C03637=1145.324,-115.065,-43.612,178.627,5.983,149.479
C03638=1145.319,-114.815,-43.621,178.630,5.984,149.478
C03639=1145.313,-114.565,-43.629,178.632,5.984,149.478
C03640=1145.308,-114.315,-43.638,178.634,5.984,149.477
C03641=1145.302,-114.066,-43.647,178.636,5.985,149.477
C03642=1145.297,-113.816,-43.655,178.637,5.985,149.476
C03643=1145.292,-113.566,-43.664,178.640,5.986,149.476
C03644=1145.286,-113.316,-43.672,178.641,5.986,149.475
C03645=1145.281,-113.066,-43.681,178.643,5.986,149.475
C03646=1145.276,-112.816,-43.690,178.646,5.987,149.474
C03647=1145.270,-112.567,-43.699,178.648,5.987,149.473
C03648=1145.265,-112.317,-43.708,178.650,5.988,149.473
C03649=1145.259,-112.068,-43.716,178.651,5.987,149.472
C03650=1145.254,-111.818,-43.725,178.654,5.988,149.472
C03651=1145.249,-111.568,-43.734,178.655,5.988,149.471
C03652=1145.244,-111.317,-43.742,178.657,5.989,149.471
C03653=1145.238,-111.068,-43.751,178.660,5.990,149.470
C03654=1145.232,-110.818,-43.760,178.661,5.990,149.470
C03655=1145.227,-110.568,-43.769,178.664,5.990,149.469
C03656=1145.222,-110.318,-43.778,178.665,5.990,149.469
C03657=1145.217,-110.069,-43.787,178.668,5.991,149.468
C03658=1145.211,-109.819,-43.796,178.669,5.991,149.468
C03659=1145.206,-109.570,-43.804,178.671,5.991,149.467
C03660=1145.200,-109.320,-43.813,178.674,5.992,149.467
C03661=1145.195,-109.070,-43.822,178.675,5.992,149.466
C03662=1145.190,-108.820,-43.831,178.678,5.992,149.466
C03663=1145.185,-108.570,-43.840,178.680,5.992,149.465
C03664=1145.179,-108.321,-43.849,178.682,5.993,149.465
C03665=1145.173,-108.071,-43.858,178.683,5.993,149.464
C03666=1145.168,-107.821,-43.867,178.685,5.994,149.464
C03667=1145.163,-107.571,-43.876,178.688,5.995,149.463
C03668=1145.158,-107.321,-43.885,178.689,5.995,149.463
C03669=1145.153,-107.071,-43.894,178.691,5.995,149.462
C03670=1145.147,-106.822,-43.902,178.694,5.995,149.462
C03671=1145.142,-106.572,-43.911,178.696,5.996,149.461
C03672=1145.136,-106.322,-43.921,178.698,5.996,149.461
C03673=1145.131,-106.072,-43.929,178.700,5.996,149.460
C03674=1145.125,-105.823,-43.938,178.702,5.997,149.460
C03675=1145.120,-105.573,-43.947,178.703,5.997,149.459
C03676=1145.115,-105.323,-43.956,178.706,5.998,149.458
C03677=1145.110,-105.073,-43.965,178.708,5.998,149.458
C03678=1145.103,-104.824,-43.974,178.710,5.998,149.457
C03679=1145.098,-104.574,-43.983,178.712,5.999,149.457
C03680=1145.093,-104.324,-43.992,178.714,5.999,149.456
C03681=1145.088,-104.074,-44.001,178.716,6.000,149.456
C03682=1145.083,-103.824,-44.010,178.718,6.000,149.455
C03683=1145.077,-103.575,-44.020,178.720,6.000,149.455
C03684=1145.072,-103.325,-44.029,178.722,6.001,149.454
C03685=1145.066,-103.052,-44.038,178.724,6.002,149.454
C03686=1145.060,-102.781,-44.048,178.727,6.001,149.453
C03687=1145.054,-102.508,-44.058,178.729,6.002,149.453
C03688=1145.049,-102.237,-44.068,178.731,6.003,149.452
C03689=1145.044,-101.987,-44.077,178.733,6.003,149.452
C03690=1145.038,-101.737,-44.086,178.735,6.003,149.451
C03691=1145.033,-101.487,-44.095,178.737,6.004,149.450
C03692=1145.027,-101.237,-44.104,178.739,6.004,149.450
C03693=1145.023,-100.988,-44.114,178.741,6.004,149.449
C03694=1145.017,-100.737,-44.123,178.743,6.005,149.449
C03695=1145.011,-100.488,-44.132,178.745,6.005,149.448
C03696=1145.006,-100.238,-44.141,178.748,6.005,149.448
C03697=1145.001,-99.989,-44.150,178.749,6.005,149.447
C03698=1144.995,-99.738,-44.159,178.751,6.006,149.447
C03699=1144.990,-99.489,-44.169,178.754,6.007,149.446
C03700=1144.985,-99.239,-44.178,178.755,6.007,149.446
C03701=1144.979,-98.989,-44.187,178.758,6.007,149.445
C03702=1144.974,-98.739,-44.196,178.760,6.008,149.445
C03703=1144.969,-98.490,-44.206,178.762,6.008,149.444
C03704=1144.963,-98.240,-44.215,178.764,6.009,149.444
C03705=1144.958,-97.990,-44.224,178.766,6.010,149.443
C03706=1144.952,-97.740,-44.233,178.768,6.010,149.443
C03707=1144.947,-97.491,-44.243,178.770,6.010,149.442
C03708=1144.942,-97.241,-44.252,178.772,6.010,149.441
C03709=1144.936,-96.991,-44.261,178.774,6.011,149.441
C03710=1144.931,-96.741,-44.270,178.776,6.011,149.441
C03711=1144.926,-96.492,-44.280,178.778,6.011,149.440
C03712=1144.921,-96.242,-44.289,178.781,6.012,149.439
C03713=1144.915,-95.992,-44.298,178.783,6.012,149.439
C03714=1144.909,-95.742,-44.307,178.784,6.012,149.438
C03715=1144.905,-95.492,-44.317,178.787,6.013,149.438
C03716=1144.899,-95.242,-44.326,178.789,6.014,149.437
C03717=1144.894,-94.992,-44.335,178.791,6.013,149.437
C03718=1144.888,-94.743,-44.346,178.793,6.014,149.436
C03719=1144.883,-94.493,-44.354,178.795,6.015,149.436
C03720=1144.878,-94.243,-44.363,178.797,6.015,149.435
C03721=1144.872,-93.994,-44.374,178.799,6.016,149.435
C03722=1144.867,-93.744,-44.382,178.801,6.015,149.434
C03723=1144.862,-93.495,-44.392,178.803,6.016,149.434
C03724=1144.856,-93.244,-44.402,178.806,6.017,149.433
C03725=1144.851,-92.995,-44.410,178.807,6.017,149.433
C03726=1144.845,-92.745,-44.421,178.809,6.018,149.432
C03727=1144.840,-92.495,-44.430,178.812,6.018,149.431
C03728=1144.834,-92.245,-44.439,178.814,6.018,149.431
C03729=1144.829,-91.996,-44.449,178.816,6.019,149.430
C03730=1144.824,-91.746,-44.458,178.818,6.019,149.430
C03731=1144.819,-91.496,-44.468,178.820,6.019,149.429
C03732=1144.813,-91.247,-44.477,178.822,6.020,149.429
C03733=1144.808,-90.997,-44.487,178.824,6.021,149.428
C03734=1144.803,-90.747,-44.496,178.826,6.020,149.428
C03735=1144.797,-90.497,-44.505,178.828,6.021,149.427
C03736=1144.792,-90.248,-44.515,178.831,6.022,149.427
C03737=1144.787,-89.997,-44.525,178.832,6.022,149.426
C03738=1144.782,-89.748,-44.534,178.835,6.022,149.426
C03739=1144.776,-89.497,-44.544,178.837,6.023,149.425
C03740=1144.771,-89.248,-44.553,178.839,6.023,149.424
C03741=1144.765,-88.998,-44.563,178.841,6.023,149.424
C03742=1144.760,-88.749,-44.573,178.843,6.024,149.423
C03743=1144.754,-88.499,-44.582,178.846,6.025,149.423
C03744=1144.749,-88.249,-44.592,178.847,6.025,149.422
C03745=1144.744,-87.999,-44.601,178.850,6.025,149.422
C03746=1144.739,-87.750,-44.611,178.852,6.026,149.421
C03747=1144.733,-87.500,-44.620,178.854,6.026,149.421
C03748=1144.729,-87.250,-44.630,178.856,6.027,149.420
C03749=1144.723,-87.000,-44.640,178.858,6.027,149.420
C03750=1144.718,-86.751,-44.649,178.860,6.027,149.419
C03751=1144.712,-86.501,-44.660,178.862,6.028,149.419
C03752=1144.707,-86.251,-44.668,178.864,6.029,149.418
C03753=1144.701,-86.002,-44.679,178.867,6.028,149.417
C03754=1144.696,-85.752,-44.688,178.869,6.029,149.417
C03755=1144.691,-85.502,-44.698,178.871,6.030,149.416
C03756=1144.686,-85.252,-44.707,178.872,6.030,149.416
C03757=1144.680,-85.002,-44.717,178.875,6.030,149.415
C03758=1144.676,-84.753,-44.727,178.877,6.031,149.415
C03759=1144.670,-84.503,-44.736,178.880,6.032,149.414
C03760=1144.664,-84.253,-44.747,178.881,6.032,149.414
C03761=1144.659,-84.003,-44.755,178.884,6.032,149.413
C03762=1144.653,-83.754,-44.766,178.886,6.033,149.413
C03763=1144.649,-83.504,-44.776,178.888,6.033,149.412
C03764=1144.643,-83.254,-44.785,178.890,6.033,149.412
C03765=1144.638,-83.004,-44.795,178.892,6.034,149.411
C03766=1144.633,-82.755,-44.805,178.894,6.034,149.410
C03767=1144.627,-82.505,-44.814,178.896,6.035,149.410
C03768=1144.622,-82.256,-44.824,178.898,6.035,149.409
C03769=1144.617,-82.005,-44.835,178.901,6.036,149.409
C03770=1144.611,-81.755,-44.844,178.903,6.036,149.408
C03771=1144.606,-81.506,-44.854,178.905,6.036,149.408
C03772=1144.601,-81.256,-44.864,178.907,6.037,149.407
C03773=1144.595,-81.006,-44.873,178.909,6.037,149.407
C03774=1144.590,-80.756,-44.883,178.911,6.038,149.406
C03775=1144.585,-80.507,-44.894,178.914,6.038,149.406
C03776=1144.579,-80.257,-44.904,178.916,6.039,149.405
C03777=1144.574,-80.007,-44.913,178.918,6.039,149.404
C03778=1144.568,-79.758,-44.923,178.920,6.039,149.404
C03779=1144.563,-79.508,-44.934,178.922,6.040,149.403
C03780=1144.559,-79.258,-44.943,178.924,6.041,149.403
C03781=1144.553,-79.008,-44.953,178.926,6.041,149.402
C03782=1144.547,-78.759,-44.963,178.929,6.041,149.402
C03783=1144.542,-78.509,-44.972,178.931,6.042,149.401
C03784=1144.537,-78.259,-44.983,178.933,6.042,149.401
C03785=1144.531,-78.009,-44.993,178.935,6.042,149.400
C03786=1144.526,-77.759,-45.003,178.937,6.043,149.400
C03787=1144.521,-77.510,-45.012,178.940,6.044,149.399
C03788=1144.515,-77.261,-45.023,178.942,6.044,149.398
C03789=1144.509,-76.989,-45.034,178.944,6.044,149.398
C03790=1144.504,-76.717,-45.044,178.946,6.045,149.397
C03791=1144.499,-76.446,-45.055,178.949,6.045,149.397
C03792=1144.492,-76.175,-45.066,178.951,6.046,149.396
C03793=1144.487,-75.925,-45.077,178.954,6.047,149.396
C03794=1144.482,-75.675,-45.086,178.955,6.047,149.395
C03795=1144.476,-75.425,-45.096,178.957,6.047,149.395
C03796=1144.471,-75.176,-45.106,178.960,6.048,149.394
C03797=1144.466,-74.926,-45.117,178.962,6.048,149.393
C03798=1144.460,-74.676,-45.127,178.964,6.048,149.393
C03799=1144.455,-74.427,-45.137,178.966,6.049,149.392
C03800=1144.450,-74.177,-45.147,178.969,6.050,149.392
C03801=1144.445,-73.927,-45.158,178.971,6.050,149.391
C03802=1144.439,-73.677,-45.168,178.972,6.050,149.391
C03803=1144.433,-73.427,-45.177,178.975,6.051,149.390
C03804=1144.429,-73.177,-45.187,178.977,6.051,149.390
C03805=1144.423,-72.928,-45.197,178.979,6.052,149.389
C03806=1144.418,-72.678,-45.208,178.982,6.053,149.389
C03807=1144.412,-72.429,-45.218,178.984,6.053,149.388
C03808=1144.407,-72.178,-45.228,178.986,6.053,149.387
C03809=1144.402,-71.929,-45.239,178.988,6.054,149.387
C03810=1144.397,-71.680,-45.248,178.991,6.055,149.386
C03811=1144.392,-71.429,-45.259,178.992,6.054,149.386
C03812=1144.386,-71.180,-45.269,178.995,6.055,149.385
C03813=1144.381,-70.930,-45.279,178.997,6.056,149.385
C03814=1144.376,-70.680,-45.290,178.999,6.056,149.384
C03815=1144.370,-70.431,-45.300,179.001,6.056,149.384
C03816=1144.364,-70.181,-45.310,179.003,6.057,149.383
C03817=1144.360,-69.931,-45.320,179.006,6.058,149.382
C03818=1144.355,-69.682,-45.330,179.008,6.058,149.382
C03819=1144.349,-69.432,-45.341,179.010,6.059,149.381
C03820=1144.344,-69.182,-45.351,179.012,6.059,149.381
C03821=1144.338,-68.932,-45.361,179.015,6.059,149.380
C03822=1144.333,-68.683,-45.372,179.017,6.060,149.380
C03823=1144.328,-68.432,-45.382,179.019,6.061,149.379
C03824=1144.322,-68.183,-45.392,179.021,6.061,149.379
C03825=1144.317,-67.933,-45.403,179.023,6.061,149.378
C03826=1144.312,-67.684,-45.414,179.025,6.062,149.378
C03827=1144.307,-67.434,-45.423,179.028,6.062,149.377
C03828=1144.302,-67.184,-45.434,179.030,6.063,149.376
C03829=1144.296,-66.935,-45.444,179.032,6.063,149.376
C03830=1144.291,-66.685,-45.454,179.035,6.064,149.375
C03831=1144.286,-66.435,-45.465,179.037,6.064,149.375
C03832=1144.280,-66.185,-45.475,179.039,6.065,149.374
C03833=1144.275,-65.935,-45.486,179.042,6.066,149.374
C03834=1144.270,-65.686,-45.496,179.043,6.066,149.373
C03835=1144.264,-65.437,-45.507,179.045,6.066,149.373
C03836=1144.259,-65.186,-45.518,179.048,6.067,149.372
C03837=1144.254,-64.937,-45.528,179.050,6.067,149.371
C03838=1144.249,-64.687,-45.538,179.052,6.068,149.371
C03839=1144.243,-64.437,-45.549,179.054,6.068,149.371
C03840=1144.238,-64.188,-45.559,179.057,6.069,149.370
C03841=1144.233,-63.938,-45.570,179.059,6.069,149.369
C03842=1144.227,-63.688,-45.580,179.061,6.070,149.369
C03843=1144.222,-63.438,-45.591,179.064,6.071,149.368
C03844=1144.217,-63.189,-45.601,179.065,6.071,149.368
C03845=1144.212,-62.938,-45.612,179.067,6.071,149.367
C03846=1144.206,-62.689,-45.623,179.070,6.072,149.366
C03847=1144.201,-62.439,-45.633,179.072,6.072,149.366
C03848=1144.196,-62.190,-45.643,179.075,6.073,149.366
C03849=1144.190,-61.940,-45.654,179.077,6.073,149.365
C03850=1144.185,-61.690,-45.665,179.079,6.074,149.364
C03851=1144.180,-61.441,-45.675,179.081,6.074,149.364
C03852=1144.175,-61.191,-45.686,179.084,6.075,149.363
C03853=1144.170,-60.942,-45.697,179.086,6.076,149.363
C03854=1144.165,-60.691,-45.707,179.088,6.076,149.362
C03855=1144.159,-60.442,-45.717,179.090,6.076,149.361
C03856=1144.154,-60.192,-45.728,179.092,6.077,149.361
C03857=1144.148,-59.942,-45.739,179.094,6.077,149.361
C03858=1144.143,-59.692,-45.750,179.097,6.078,149.360
C03859=1144.137,-59.443,-45.760,179.099,6.079,149.359
C03860=1144.133,-59.193,-45.771,179.102,6.079,149.359
C03861=1144.127,-58.943,-45.782,179.104,6.079,149.358
C03862=1144.122,-58.693,-45.792,179.106,6.080,149.358
C03863=1144.117,-58.444,-45.803,179.108,6.081,149.357
C03864=1144.112,-58.194,-45.814,179.111,6.081,149.356
C03865=1144.106,-57.945,-45.824,179.113,6.082,149.356
C03866=1144.101,-57.695,-45.835,179.115,6.082,149.356
C03867=1144.095,-57.445,-45.846,179.117,6.082,149.355
C03868=1144.090,-57.195,-45.857,179.119,6.083,149.354
C03869=1144.085,-56.946,-45.868,179.121,6.084,149.354
C03870=1144.080,-56.696,-45.878,179.124,6.084,149.353
C03871=1144.075,-56.446,-45.889,179.126,6.085,149.353
C03872=1144.070,-56.196,-45.900,179.129,6.086,149.352
C03873=1144.065,-55.947,-45.911,179.131,6.086,149.351
C03874=1144.059,-55.697,-45.922,179.133,6.086,149.351
C03875=1144.054,-55.447,-45.933,179.135,6.087,149.351
C03876=1144.048,-55.198,-45.943,179.138,6.087,149.350
C03877=1144.044,-54.948,-45.954,179.140,6.088,149.349
C03878=1144.038,-54.699,-45.965,179.142,6.089,149.349
C03879=1144.033,-54.448,-45.975,179.145,6.089,149.348
C03880=1144.028,-54.198,-45.987,179.147,6.090,149.348
C03881=1144.022,-53.949,-45.997,179.148,6.090,149.347
C03882=1144.017,-53.699,-46.009,179.151,6.090,149.347
C03883=1144.012,-53.450,-46.019,179.153,6.091,149.346
C03884=1144.006,-53.200,-46.031,179.156,6.092,149.346
C03885=1144.001,-52.950,-46.041,179.158,6.092,149.345
C03886=1143.996,-52.701,-46.052,179.160,6.093,149.344
C03887=1143.991,-52.451,-46.064,179.163,6.094,149.344
C03888=1143.986,-52.201,-46.074,179.165,6.093,149.343
C03889=1143.980,-51.952,-46.086,179.167,6.094,149.343
C03890=1143.975,-51.702,-46.096,179.169,6.095,149.342
C03891=1143.970,-51.452,-46.107,179.172,6.095,149.342
C03892=1143.964,-51.202,-46.118,179.174,6.096,149.341
C03893=1143.959,-50.932,-46.130,179.177,6.096,149.340
C03894=1143.953,-50.661,-46.142,179.179,6.097,149.340
C03895=1143.947,-50.390,-46.154,179.181,6.098,149.339
C03896=1143.941,-50.120,-46.166,179.184,6.098,149.339
C03897=1143.937,-49.870,-46.177,179.186,6.099,149.338
C03898=1143.931,-49.620,-46.187,179.188,6.100,149.338
C03899=1143.926,-49.371,-46.199,179.191,6.100,149.337
C03900=1143.921,-49.121,-46.211,179.193,6.101,149.336
C03901=1143.915,-48.871,-46.221,179.195,6.101,149.336
C03902=1143.910,-48.621,-46.233,179.197,6.101,149.335
C03903=1143.905,-48.372,-46.244,179.200,6.102,149.335
C03904=1143.900,-48.122,-46.254,179.202,6.103,149.334
C03905=1143.894,-47.872,-46.266,179.204,6.103,149.334
C03906=1143.889,-47.623,-46.277,179.207,6.104,149.333
C03907=1143.884,-47.373,-46.288,179.209,6.105,149.333
C03908=1143.878,-47.123,-46.300,179.212,6.105,149.332
C03909=1143.874,-46.874,-46.311,179.214,6.106,149.331
C03910=1143.868,-46.624,-46.321,179.216,6.107,149.331
C03911=1143.863,-46.374,-46.333,179.219,6.107,149.330
C03912=1143.858,-46.124,-46.344,179.220,6.107,149.330
C03913=1143.852,-45.875,-46.355,179.222,6.108,149.329
C03914=1143.847,-45.625,-46.366,179.225,6.108,149.329
C03915=1143.842,-45.375,-46.378,179.227,6.109,149.328
C03916=1143.836,-45.126,-46.389,179.230,6.110,149.328
C03917=1143.831,-44.876,-46.400,179.232,6.110,149.327
C03918=1143.826,-44.626,-46.412,179.234,6.111,149.326
C03919=1143.821,-44.376,-46.423,179.237,6.111,149.326
C03920=1143.816,-44.127,-46.434,179.239,6.112,149.325
C03921=1143.810,-43.877,-46.446,179.241,6.113,149.325
C03922=1143.805,-43.627,-46.456,179.244,6.113,149.324
C03923=1143.799,-43.378,-46.468,179.246,6.113,149.324
C03924=1143.795,-43.128,-46.479,179.248,6.114,149.323
C03925=1143.789,-42.878,-46.491,179.250,6.114,149.322
C03926=1143.785,-42.629,-46.502,179.253,6.115,149.322
C03927=1143.778,-42.380,-46.514,179.255,6.116,149.321
C03928=1143.773,-42.129,-46.524,179.258,6.116,149.321
C03929=1143.769,-41.880,-46.536,179.260,6.117,149.320
C03930=1143.763,-41.630,-46.547,179.262,6.118,149.320
C03931=1143.758,-41.381,-46.558,179.265,6.118,149.319
C03932=1143.753,-41.131,-46.570,179.267,6.119,149.319
C03933=1143.748,-40.881,-46.582,179.269,6.120,149.318
C03934=1143.743,-40.631,-46.593,179.272,6.120,149.317
C03935=1143.737,-40.382,-46.604,179.274,6.121,149.317
C03936=1143.731,-40.132,-46.616,179.276,6.121,149.316
C03937=1143.727,-39.882,-46.627,179.279,6.122,149.316
C03938=1143.721,-39.632,-46.639,179.281,6.122,149.315
C03939=1143.716,-39.382,-46.651,179.283,6.123,149.315
C03940=1143.711,-39.133,-46.662,179.285,6.123,149.314
C03941=1143.705,-38.883,-46.673,179.288,6.124,149.313
C03942=1143.701,-38.634,-46.685,179.290,6.125,149.313
C03943=1143.695,-38.384,-46.697,179.292,6.125,149.312
C03944=1143.690,-38.134,-46.708,179.295,6.126,149.312
C03945=1143.684,-37.885,-46.719,179.297,6.127,149.311
C03946=1143.680,-37.635,-46.731,179.300,6.127,149.311
C03947=1143.674,-37.385,-46.743,179.302,6.128,149.310
C03948=1143.669,-37.136,-46.754,179.304,6.129,149.310
C03949=1143.664,-36.886,-46.766,179.307,6.129,149.309
C03950=1143.658,-36.637,-46.777,179.309,6.130,149.308
C03951=1143.653,-36.387,-46.789,179.311,6.131,149.308
C03952=1143.648,-36.137,-46.800,179.314,6.131,149.307
C03953=1143.643,-35.887,-46.812,179.316,6.132,149.307
C03954=1143.638,-35.638,-46.824,179.319,6.132,149.306
C03955=1143.632,-35.388,-46.836,179.321,6.133,149.306
C03956=1143.627,-35.139,-46.846,179.323,6.134,149.305
C03957=1143.622,-34.889,-46.858,179.326,6.134,149.304
C03958=1143.616,-34.639,-46.870,179.328,6.135,149.304
C03959=1143.612,-34.389,-46.882,179.330,6.135,149.303
C03960=1143.606,-34.140,-46.894,179.333,6.136,149.303
C03961=1143.601,-33.890,-46.906,179.335,6.137,149.302
C03962=1143.596,-33.640,-46.917,179.337,6.137,149.302
C03963=1143.590,-33.391,-46.929,179.340,6.138,149.301
C03964=1143.585,-33.141,-46.941,179.342,6.139,149.301
C03965=1143.580,-32.892,-46.952,179.344,6.138,149.300
C03966=1143.575,-32.642,-46.964,179.346,6.139,149.300
C03967=1143.569,-32.392,-46.976,179.349,6.140,149.299
C03968=1143.565,-32.143,-46.988,179.351,6.140,149.298
C03969=1143.560,-31.893,-47.000,179.353,6.141,149.298
C03970=1143.554,-31.643,-47.012,179.356,6.142,149.297
C03971=1143.549,-31.393,-47.023,179.358,6.142,149.297
C03972=1143.544,-31.143,-47.035,179.361,6.143,149.296
C03973=1143.538,-30.895,-47.047,179.363,6.144,149.296
C03974=1143.533,-30.645,-47.059,179.365,6.144,149.295
C03975=1143.528,-30.395,-47.070,179.368,6.145,149.294
C03976=1143.523,-30.145,-47.082,179.370,6.146,149.294
C03977=1143.517,-29.895,-47.094,179.373,6.146,149.293
C03978=1143.512,-29.646,-47.106,179.375,6.147,149.293
C03979=1143.507,-29.396,-47.118,179.377,6.148,149.292
C03980=1143.502,-29.146,-47.130,179.380,6.148,149.292
C03981=1143.497,-28.896,-47.142,179.382,6.149,149.291
C03982=1143.491,-28.647,-47.154,179.384,6.150,149.291
C03983=1143.487,-28.397,-47.165,179.387,6.150,149.290
C03984=1143.481,-28.147,-47.177,179.389,6.151,149.289
C03985=1143.476,-27.898,-47.190,179.391,6.151,149.289
C03986=1143.471,-27.648,-47.202,179.394,6.152,149.288
C03987=1143.465,-27.398,-47.214,179.396,6.153,149.288
C03988=1143.461,-27.149,-47.226,179.399,6.154,149.287
C03989=1143.456,-26.899,-47.238,179.401,6.155,149.287
C03990=1143.450,-26.649,-47.249,179.404,6.155,149.286
C03991=1143.445,-26.400,-47.262,179.406,6.156,149.285
C03992=1143.440,-26.150,-47.274,179.408,6.157,149.285
C03993=1143.435,-25.901,-47.285,179.411,6.157,149.284
C03994=1143.430,-25.651,-47.298,179.413,6.158,149.284
C03995=1143.424,-25.401,-47.310,179.416,6.158,149.283
C03996=1143.419,-25.151,-47.322,179.418,6.159,149.283
C03997=1143.413,-24.882,-47.335,179.421,6.160,149.282
C03998=1143.408,-24.612,-47.348,179.423,6.160,149.281
C03999=1143.401,-24.342,-47.361,179.425,6.161,149.281
C04000=1143.396,-24.072,-47.374,179.428,6.162,149.280
C04001=1143.391,-23.822,-47.387,179.431,6.163,149.280
C04002=1143.385,-23.572,-47.399,179.433,6.164,149.279
C04003=1143.381,-23.323,-47.410,179.436,6.164,149.278
C04004=1143.376,-23.073,-47.422,179.438,6.165,149.278
C04005=1143.370,-22.824,-47.434,179.440,6.166,149.277
C04006=1143.365,-22.574,-47.447,179.443,6.166,149.277
C04007=1143.360,-22.324,-47.459,179.445,6.167,149.276
C04008=1143.355,-22.075,-47.471,179.448,6.167,149.276
C04009=1143.349,-21.825,-47.483,179.450,6.168,149.275
C04010=1143.344,-21.576,-47.496,179.452,6.169,149.275
C04011=1143.339,-21.325,-47.508,179.455,6.169,149.274
C04012=1143.334,-21.076,-47.521,179.457,6.170,149.273
C04013=1143.329,-20.826,-47.533,179.460,6.170,149.273
C04014=1143.323,-20.576,-47.545,179.462,6.171,149.272
C04015=1143.318,-20.327,-47.557,179.464,6.172,149.272
C04016=1143.313,-20.077,-47.570,179.467,6.172,149.271
C04017=1143.308,-19.828,-47.582,179.469,6.173,149.271
C04018=1143.302,-19.578,-47.594,179.471,6.174,149.270
C04019=1143.297,-19.329,-47.607,179.474,6.174,149.270
C04020=1143.292,-19.079,-47.619,179.476,6.176,149.269
C04021=1143.287,-18.829,-47.631,179.479,6.176,149.268
C04022=1143.281,-18.579,-47.643,179.481,6.177,149.268
C04023=1143.277,-18.329,-47.656,179.484,6.178,149.267
C04024=1143.272,-18.080,-47.669,179.486,6.178,149.267
C04025=1143.266,-17.830,-47.681,179.488,6.179,149.266
C04026=1143.261,-17.581,-47.693,179.491,6.180,149.266
C04027=1143.256,-17.332,-47.706,179.493,6.181,149.265
C04028=1143.251,-17.082,-47.718,179.496,6.181,149.264
C04029=1143.245,-16.832,-47.730,179.498,6.182,149.264
C04030=1143.240,-16.582,-47.742,179.500,6.183,149.263
C04031=1143.235,-16.332,-47.755,179.503,6.183,149.263
C04032=1143.230,-16.083,-47.768,179.505,6.184,149.262
C04033=1143.225,-15.834,-47.780,179.508,6.185,149.262
C04034=1143.220,-15.584,-47.792,179.510,6.186,149.261
C04035=1143.215,-15.334,-47.805,179.513,6.187,149.261
C04036=1143.210,-15.085,-47.817,179.515,6.187,149.260
C04037=1143.204,-14.835,-47.829,179.517,6.188,149.259
C04038=1143.200,-14.585,-47.842,179.520,6.188,149.259
C04039=1143.194,-14.336,-47.855,179.522,6.189,149.258
C04040=1143.189,-14.086,-47.868,179.524,6.190,149.258
C04041=1143.183,-13.836,-47.880,179.527,6.190,149.257
C04042=1143.178,-13.587,-47.893,179.529,6.191,149.257
C04043=1143.173,-13.337,-47.906,179.532,6.191,149.256
C04044=1143.168,-13.088,-47.918,179.535,6.193,149.256
C04045=1143.163,-12.838,-47.930,179.537,6.194,149.255
C04046=1143.158,-12.588,-47.943,179.540,6.194,149.254
C04047=1143.152,-12.339,-47.956,179.542,6.195,149.254
C04048=1143.147,-12.089,-47.969,179.544,6.195,149.253
C04049=1143.142,-11.839,-47.981,179.547,6.196,149.253
C04050=1143.137,-11.590,-47.994,179.549,6.197,149.252
C04051=1143.132,-11.340,-48.006,179.551,6.197,149.252
C04052=1143.127,-11.091,-48.018,179.554,6.198,149.251
C04053=1143.121,-10.841,-48.032,179.557,6.200,149.250
C04054=1143.116,-10.591,-48.045,179.559,6.200,149.250
C04055=1143.111,-10.342,-48.057,179.561,6.201,149.249
C04056=1143.106,-10.093,-48.070,179.564,6.202,149.249
C04057=1143.101,-9.843,-48.083,179.566,6.202,149.248
C04058=1143.095,-9.592,-48.095,179.569,6.203,149.248
C04059=1143.090,-9.343,-48.108,179.571,6.204,149.247
C04060=1143.085,-9.094,-48.120,179.573,6.204,149.246
C04061=1143.081,-8.844,-48.133,179.576,6.206,149.246
C04062=1143.075,-8.594,-48.146,179.578,6.206,149.246
C04063=1143.070,-8.345,-48.159,179.581,6.207,149.245
C04064=1143.064,-8.095,-48.172,179.583,6.208,149.244
C04065=1143.060,-7.845,-48.185,179.586,6.208,149.244
C04066=1143.055,-7.596,-48.197,179.588,6.209,149.243
C04067=1143.049,-7.346,-48.211,179.590,6.210,149.243
C04068=1143.044,-7.096,-48.224,179.594,6.211,149.242
C04069=1143.039,-6.847,-48.236,179.596,6.212,149.242
C04070=1143.034,-6.598,-48.249,179.598,6.212,149.241
C04071=1143.028,-6.348,-48.262,179.601,6.213,149.240
C04072=1143.024,-6.098,-48.275,179.603,6.214,149.240
C04073=1143.019,-5.849,-48.288,179.605,6.214,149.239
C04074=1143.013,-5.599,-48.301,179.608,6.215,149.239
C04075=1143.008,-5.349,-48.314,179.611,6.216,149.238
C04076=1143.003,-5.100,-48.326,179.613,6.217,149.238
C04077=1142.997,-4.850,-48.340,179.615,6.218,149.237
C04078=1142.993,-4.600,-48.352,179.618,6.218,149.237
C04079=1142.988,-4.351,-48.365,179.620,6.219,149.236
C04080=1142.982,-4.101,-48.378,179.623,6.219,149.235
C04081=1142.977,-3.851,-48.391,179.625,6.221,149.235
C04082=1142.972,-3.603,-48.405,179.628,6.221,149.234
C04083=1142.967,-3.353,-48.418,179.630,6.222,149.234
C04084=1142.962,-3.103,-48.431,179.632,6.223,149.233
C04085=1142.956,-2.853,-48.444,179.635,6.223,149.233
C04086=1142.951,-2.604,-48.457,179.637,6.224,149.232
C04087=1142.947,-2.354,-48.469,179.641,6.226,149.231
C04088=1142.941,-2.104,-48.483,179.643,6.226,149.231
C04089=1142.936,-1.854,-48.496,179.645,6.227,149.230
C04090=1142.931,-1.606,-48.509,179.648,6.228,149.230
C04091=1142.925,-1.356,-48.522,179.650,6.228,149.229
C04092=1142.921,-1.106,-48.535,179.652,6.229,149.229
C04093=1142.915,-0.856,-48.548,179.655,6.230,149.228
C04094=1142.910,-0.607,-48.561,179.657,6.231,149.228
C04095=1142.905,-0.357,-48.575,179.660,6.232,149.227
C04096=1142.900,-0.108,-48.588,179.662,6.232,149.227
C04097=1142.895,0.142,-48.601,179.665,6.233,149.226
C04098=1142.889,0.392,-48.614,179.668,6.234,149.225
C04099=1142.885,0.640,-48.627,179.670,6.235,149.225
C04100=1142.879,0.891,-48.641,179.672,6.236,149.224
C04101=1142.874,1.161,-48.655,179.675,6.237,149.224
C04102=1142.868,1.429,-48.669,179.678,6.238,149.223
C04103=1142.863,1.699,-48.683,179.681,6.238,149.222
C04104=1142.857,1.969,-48.698,179.683,6.239,149.222
C04105=1142.852,2.218,-48.711,179.686,6.240,149.221
C04106=1142.847,2.468,-48.725,179.688,6.241,149.221
C04107=1142.842,2.717,-48.738,179.690,6.242,149.220
C04108=1142.836,2.967,-48.751,179.693,6.242,149.220
C04109=1142.832,3.217,-48.764,179.695,6.243,149.219
C04110=1142.826,3.466,-48.778,179.698,6.244,149.218
C04111=1142.822,3.716,-48.791,179.701,6.245,149.218
C04112=1142.816,3.965,-48.804,179.703,6.246,149.217
C04113=1142.811,4.215,-48.818,179.705,6.246,149.217
C04114=1142.806,4.464,-48.831,179.708,6.247,149.216
C04115=1142.801,4.714,-48.844,179.711,6.248,149.216
C04116=1142.796,4.963,-48.858,179.713,6.249,149.215
C04117=1142.790,5.214,-48.871,179.716,6.250,149.215
C04118=1142.785,5.462,-48.885,179.718,6.250,149.214
C04119=1142.780,5.713,-48.898,179.721,6.252,149.214
C04120=1142.775,5.962,-48.911,179.723,6.253,149.213
C04121=1142.770,6.212,-48.925,179.725,6.253,149.212
C04122=1142.764,6.461,-48.938,179.728,6.254,149.212
C04123=1142.760,6.711,-48.952,179.730,6.255,149.211
C04124=1142.754,6.960,-48.965,179.733,6.256,149.211
C04125=1142.750,7.210,-48.979,179.736,6.257,149.210
C04126=1142.744,7.459,-48.992,179.738,6.257,149.210
C04127=1142.739,7.709,-49.006,179.741,6.258,149.209
C04128=1142.734,7.958,-49.019,179.743,6.259,149.209
C04129=1142.729,8.208,-49.033,179.745,6.260,149.208
C04130=1142.723,8.458,-49.047,179.748,6.261,149.207
C04131=1142.719,8.707,-49.060,179.750,6.262,149.207
C04132=1142.714,8.958,-49.074,179.754,6.263,149.206
C04133=1142.708,9.207,-49.088,179.756,6.264,149.206
C04134=1142.704,9.457,-49.101,179.758,6.264,149.205
C04135=1142.698,9.706,-49.115,179.761,6.265,149.205
C04136=1142.693,9.955,-49.129,179.763,6.266,149.204
C04137=1142.688,10.205,-49.141,179.766,6.267,149.204
C04138=1142.683,10.454,-49.156,179.768,6.268,149.203
C04139=1142.678,10.705,-49.169,179.770,6.269,149.203
C04140=1142.673,10.953,-49.183,179.774,6.270,149.202
C04141=1142.668,11.204,-49.196,179.776,6.271,149.201
C04142=1142.662,11.453,-49.210,179.778,6.271,149.201
C04143=1142.657,11.702,-49.224,179.781,6.272,149.200
C04144=1142.652,11.952,-49.237,179.784,6.273,149.200
C04145=1142.647,12.201,-49.251,179.786,6.274,149.199
C04146=1142.642,12.451,-49.265,179.788,6.275,149.199
C04147=1142.636,12.701,-49.279,179.791,6.275,149.198
C04148=1142.632,12.950,-49.292,179.794,6.277,149.198
C04149=1142.627,13.200,-49.307,179.796,6.277,149.197
C04150=1142.621,13.449,-49.320,179.798,6.278,149.196
C04151=1142.616,13.699,-49.334,179.801,6.280,149.196
C04152=1142.611,13.948,-49.348,179.804,6.280,149.195
C04153=1142.607,14.198,-49.362,179.806,6.281,149.195
C04154=1142.601,14.448,-49.375,179.809,6.281,149.194
C04155=1142.596,14.697,-49.389,179.811,6.283,149.194
C04156=1142.591,14.947,-49.403,179.814,6.284,149.193
C04157=1142.586,15.196,-49.418,179.816,6.284,149.193
C04158=1142.581,15.446,-49.430,179.819,6.286,149.192
C04159=1142.576,15.695,-49.445,179.822,6.286,149.191
C04160=1142.571,15.945,-49.459,179.824,6.287,149.191
C04161=1142.565,16.194,-49.473,179.826,6.288,149.190
C04162=1142.560,16.444,-49.486,179.829,6.289,149.190
C04163=1142.555,16.694,-49.501,179.831,6.290,149.189
C04164=1142.550,16.943,-49.514,179.834,6.290,149.189
C04165=1142.545,17.193,-49.528,179.837,6.292,149.188
C04166=1142.540,17.442,-49.542,179.839,6.293,149.188
C04167=1142.535,17.691,-49.556,179.842,6.293,149.187
C04168=1142.529,17.942,-49.570,179.844,6.295,149.187
C04169=1142.525,18.191,-49.584,179.847,6.295,149.186
C04170=1142.520,18.441,-49.599,179.849,6.296,149.185
C04171=1142.514,18.690,-49.612,179.851,6.297,149.185
C04172=1142.509,18.940,-49.627,179.855,6.298,149.184
C04173=1142.504,19.189,-49.641,179.857,6.299,149.184
C04174=1142.499,19.438,-49.654,179.860,6.299,149.183
C04175=1142.494,19.688,-49.669,179.862,6.301,149.183
C04176=1142.489,19.938,-49.683,179.864,6.302,149.182
C04177=1142.484,20.187,-49.697,179.867,6.302,149.182
C04178=1142.479,20.437,-49.710,179.870,6.304,149.181
C04179=1142.474,20.687,-49.725,179.873,6.304,149.180
C04180=1142.469,20.936,-49.739,179.875,6.305,149.180
C04181=1142.464,21.186,-49.753,179.877,6.307,149.180
C04182=1142.458,21.435,-49.767,179.880,6.307,149.179
C04183=1142.453,21.685,-49.781,179.882,6.308,149.178
C04184=1142.448,21.934,-49.796,179.885,6.310,149.178
C04185=1142.443,22.184,-49.810,179.888,6.310,149.177
C04186=1142.438,22.433,-49.824,179.890,6.311,149.177
C04187=1142.433,22.683,-49.838,179.893,6.312,149.176
C04188=1142.428,22.933,-49.852,179.895,6.313,149.176
C04189=1142.423,23.182,-49.867,179.897,6.314,149.175
C04190=1142.418,23.431,-49.882,179.901,6.315,149.175
C04191=1142.413,23.680,-49.896,179.903,6.316,149.174
C04192=1142.408,23.930,-49.910,179.906,6.316,149.173
C04193=1142.403,24.180,-49.924,179.908,6.318,149.173
C04194=1142.398,24.430,-49.938,179.910,6.319,149.172
C04195=1142.393,24.679,-49.953,179.913,6.319,149.172
C04196=1142.387,24.928,-49.967,179.916,6.321,149.171
C04197=1142.382,25.178,-49.981,179.919,6.321,149.171
C04198=1142.377,25.428,-49.996,179.921,6.322,149.170
C04199=1142.372,25.678,-50.010,179.923,6.324,149.170
C04200=1142.367,25.927,-50.025,179.926,6.324,149.169
C04201=1142.362,26.177,-50.039,179.928,6.325,149.169
C04202=1142.357,26.426,-50.053,179.931,6.326,149.168
C04203=1142.352,26.675,-50.067,179.934,6.327,149.167
C04204=1142.347,26.925,-50.082,179.936,6.329,149.167
C04205=1142.341,27.194,-50.097,179.939,6.329,149.166
C04206=1142.336,27.463,-50.114,179.942,6.331,149.166
C04207=1142.330,27.732,-50.129,179.944,6.331,149.165
C04208=1142.325,28.001,-50.144,179.948,6.333,149.165
C04209=1142.320,28.251,-50.159,179.950,6.333,149.164
C04210=1142.314,28.500,-50.173,179.953,6.335,149.164
C04211=1142.309,28.749,-50.188,179.955,6.335,149.163
C04212=1142.304,28.999,-50.202,179.957,6.336,149.162
C04213=1142.299,29.249,-50.217,179.961,6.338,149.162
C04214=1142.295,29.498,-50.232,179.963,6.338,149.161
C04215=1142.290,29.747,-50.246,179.965,6.339,149.161
C04216=1142.284,29.997,-50.261,179.968,6.340,149.160
C04217=1142.279,30.247,-50.275,179.970,6.341,149.160
C04218=1142.274,30.496,-50.290,179.973,6.343,149.159
C04219=1142.269,30.746,-50.304,179.976,6.343,149.159
C04220=1142.264,30.995,-50.318,179.978,6.344,149.158
C04221=1142.258,31.244,-50.334,179.981,6.345,149.158
C04222=1142.253,31.494,-50.348,179.983,6.346,149.157
C04223=1142.249,31.744,-50.363,179.986,6.348,149.157
C04224=1142.244,31.993,-50.378,179.989,6.348,149.156
C04225=1142.238,32.243,-50.392,179.991,6.349,149.155
C04226=1142.234,32.492,-50.407,179.994,6.351,149.155
C04227=1142.229,32.742,-50.422,179.996,6.351,149.154
C04228=1142.224,32.991,-50.436,179.999,6.353,149.154
C04229=1142.218,33.241,-50.452,-179.998,6.353,149.153
C04230=1142.213,33.490,-50.466,-179.996,6.354,149.153
C04231=1142.209,33.740,-50.481,-179.993,6.356,149.152
C04232=1142.203,33.990,-50.496,-179.991,6.356,149.152
C04233=1142.198,34.239,-50.511,-179.988,6.358,149.151
C04234=1142.193,34.488,-50.525,-179.985,6.358,149.151
C04235=1142.188,34.738,-50.540,-179.983,6.359,149.150
C04236=1142.183,34.988,-50.555,-179.980,6.361,149.150
C04237=1142.178,35.237,-50.569,-179.978,6.361,149.149
C04238=1142.173,35.487,-50.585,-179.975,6.363,149.148
C04239=1142.168,35.736,-50.599,-179.973,6.364,149.148
C04240=1142.163,35.985,-50.614,-179.969,6.365,149.147
C04241=1142.158,36.235,-50.630,-179.967,6.366,149.147
C04242=1142.153,36.485,-50.644,-179.965,6.366,149.146
C04243=1142.148,36.734,-50.659,-179.962,6.368,149.146
C04244=1142.142,36.984,-50.674,-179.960,6.369,149.145
C04245=1142.138,37.233,-50.689,-179.956,6.370,149.145
C04246=1142.132,37.483,-50.704,-179.954,6.371,149.144
C04247=1142.127,37.732,-50.719,-179.952,6.372,149.144
C04248=1142.122,37.982,-50.733,-179.949,6.373,149.143
C04249=1142.117,38.231,-50.748,-179.946,6.375,149.143
C04250=1142.112,38.480,-50.763,-179.944,6.375,149.142
C04251=1142.107,38.730,-50.778,-179.941,6.376,149.142
C04252=1142.102,38.979,-50.793,-179.939,6.377,149.141
C04253=1142.097,39.229,-50.809,-179.936,6.378,149.140
C04254=1142.092,39.478,-50.823,-179.933,6.380,149.140
C04255=1142.086,39.728,-50.839,-179.931,6.380,149.140
C04256=1142.082,39.977,-50.854,-179.928,6.382,149.139
C04257=1142.077,40.227,-50.868,-179.926,6.382,149.138
C04258=1142.072,40.477,-50.884,-179.923,6.384,149.138
C04259=1142.067,40.726,-50.899,-179.920,6.385,149.137
C04260=1142.062,40.976,-50.914,-179.917,6.386,149.137
C04261=1142.057,41.225,-50.929,-179.915,6.387,149.136
C04262=1142.052,41.474,-50.944,-179.913,6.387,149.136
C04263=1142.047,41.724,-50.959,-179.910,6.389,149.135
C04264=1142.041,41.973,-50.974,-179.907,6.390,149.135
C04265=1142.037,42.222,-50.989,-179.904,6.391,149.134
C04266=1142.032,42.473,-51.005,-179.902,6.392,149.134
C04267=1142.026,42.722,-51.021,-179.899,6.393,149.133
C04268=1142.021,42.972,-51.035,-179.897,6.394,149.133
C04269=1142.016,43.221,-51.051,-179.894,6.396,149.132
C04270=1142.011,43.470,-51.066,-179.891,6.396,149.131
C04271=1142.006,43.720,-51.081,-179.889,6.398,149.131
C04272=1142.001,43.969,-51.096,-179.887,6.399,149.131
C04273=1141.996,44.219,-51.111,-179.883,6.400,149.130
C04274=1141.992,44.468,-51.126,-179.881,6.401,149.129
C04275=1141.986,44.718,-51.142,-179.878,6.402,149.129
C04276=1141.981,44.967,-51.158,-179.876,6.403,149.128
C04277=1141.976,45.216,-51.173,-179.873,6.405,149.128
C04278=1141.971,45.466,-51.188,-179.870,6.405,149.127
C04279=1141.967,45.716,-51.204,-179.868,6.407,149.127
C04280=1141.961,45.966,-51.218,-179.865,6.408,149.126
C04281=1141.956,46.215,-51.234,-179.862,6.409,149.126
C04282=1141.951,46.464,-51.249,-179.860,6.410,149.125
C04283=1141.946,46.713,-51.265,-179.857,6.411,149.125
C04284=1141.941,46.964,-51.281,-179.855,6.412,149.124
C04285=1141.936,47.213,-51.296,-179.852,6.413,149.124
C04286=1141.931,47.462,-51.311,-179.850,6.414,149.123
C04287=1141.925,47.711,-51.327,-179.846,6.415,149.123
C04288=1141.921,47.961,-51.342,-179.844,6.416,149.122
C04289=1141.916,48.211,-51.358,-179.842,6.418,149.122
C04290=1141.911,48.460,-51.373,-179.839,6.418,149.121
C04291=1141.906,48.709,-51.388,-179.836,6.420,149.121
C04292=1141.901,48.959,-51.404,-179.834,6.421,149.120
C04293=1141.896,49.209,-51.420,-179.831,6.422,149.119
C04294=1141.891,49.458,-51.435,-179.829,6.423,149.119
C04295=1141.886,49.707,-51.450,-179.826,6.425,149.119
C04296=1141.880,49.957,-51.466,-179.823,6.425,149.118
C04297=1141.876,50.206,-51.481,-179.820,6.427,149.117
C04298=1141.871,50.456,-51.497,-179.818,6.427,149.117
C04299=1141.866,50.705,-51.512,-179.815,6.429,149.116
C04300=1141.860,50.955,-51.528,-179.813,6.430,149.116
C04301=1141.856,51.204,-51.544,-179.810,6.431,149.115
C04302=1141.851,51.453,-51.560,-179.808,6.432,149.115
C04303=1141.846,51.702,-51.575,-179.805,6.433,149.114
C04304=1141.841,51.953,-51.591,-179.802,6.435,149.114
C04305=1141.835,52.202,-51.607,-179.799,6.436,149.113
C04306=1141.831,52.451,-51.622,-179.797,6.437,149.113
C04307=1141.825,52.700,-51.637,-179.794,6.438,149.112
C04308=1141.821,52.951,-51.653,-179.791,6.439,149.112
C04309=1141.815,53.219,-51.670,-179.789,6.440,149.111
C04310=1141.810,53.488,-51.687,-179.786,6.441,149.111
C04311=1141.804,53.756,-51.704,-179.783,6.443,149.110
C04312=1141.798,54.025,-51.721,-179.780,6.444,149.109
C04313=1141.794,54.274,-51.737,-179.778,6.445,149.109
C04314=1141.789,54.523,-51.753,-179.774,6.446,149.108
C04315=1141.784,54.772,-51.769,-179.772,6.447,149.108
C04316=1141.779,55.023,-51.785,-179.770,6.449,149.107
C04317=1141.774,55.272,-51.800,-179.766,6.450,149.107
C04318=1141.769,55.521,-51.817,-179.764,6.451,149.106
C04319=1141.764,55.771,-51.833,-179.761,6.453,149.106
C04320=1141.759,56.020,-51.848,-179.759,6.453,149.105
C04321=1141.754,56.270,-51.863,-179.756,6.455,149.105
C04322=1141.749,56.519,-51.880,-179.754,6.456,149.104
C04323=1141.744,56.768,-51.895,-179.751,6.457,149.104
C04324=1141.739,57.018,-51.911,-179.748,6.459,149.103
C04325=1141.734,57.267,-51.928,-179.746,6.459,149.103
C04326=1141.729,57.517,-51.944,-179.742,6.461,149.102
C04327=1141.724,57.767,-51.959,-179.740,6.462,149.102
C04328=1141.719,58.015,-51.975,-179.738,6.463,149.101
C04329=1141.714,58.266,-51.991,-179.735,6.464,149.101
C04330=1141.709,58.514,-52.008,-179.732,6.465,149.100
C04331=1141.704,58.764,-52.024,-179.729,6.467,149.100
C04332=1141.699,59.014,-52.039,-179.727,6.468,149.099
C04333=1141.694,59.263,-52.056,-179.724,6.469,149.099
C04334=1141.689,59.513,-52.072,-179.722,6.470,149.098
C04335=1141.684,59.762,-52.088,-179.719,6.472,149.098
C04336=1141.679,60.012,-52.104,-179.716,6.473,149.097
C04337=1141.674,60.260,-52.120,-179.714,6.474,149.097
C04338=1141.669,60.511,-52.136,-179.711,6.475,149.096
C04339=1141.664,60.760,-52.152,-179.708,6.476,149.095
C04340=1141.659,61.009,-52.168,-179.706,6.477,149.095
C04341=1141.654,61.259,-52.184,-179.703,6.479,149.095
C04342=1141.649,61.508,-52.200,-179.700,6.480,149.094
C04343=1141.644,61.758,-52.216,-179.697,6.481,149.094
C04344=1141.639,62.006,-52.232,-179.695,6.482,149.093
C04345=1141.635,62.256,-52.249,-179.693,6.484,149.093
C04346=1141.629,62.505,-52.265,-179.689,6.485,149.092
C04347=1141.625,62.755,-52.281,-179.687,6.486,149.092
C04348=1141.619,63.004,-52.297,-179.684,6.488,149.091
C04349=1141.615,63.254,-52.314,-179.682,6.488,149.090
C04350=1141.609,63.503,-52.329,-179.679,6.490,149.090
C04351=1141.605,63.753,-52.346,-179.676,6.491,149.090
C04352=1141.599,64.002,-52.363,-179.674,6.492,149.089
C04353=1141.594,64.252,-52.379,-179.671,6.493,149.088
C04354=1141.589,64.501,-52.395,-179.668,6.495,149.088
C04355=1141.584,64.751,-52.411,-179.666,6.496,149.087
C04356=1141.579,64.999,-52.427,-179.663,6.497,149.087
C04357=1141.575,65.249,-52.444,-179.660,6.499,149.087
C04358=1141.570,65.499,-52.460,-179.658,6.500,149.086
C04359=1141.564,65.748,-52.477,-179.655,6.501,149.085
C04360=1141.560,65.998,-52.493,-179.652,6.502,149.085
C04361=1141.554,66.247,-52.509,-179.650,6.503,149.085
C04362=1141.550,66.497,-52.526,-179.646,6.505,149.084
C04363=1141.545,66.745,-52.542,-179.644,6.506,149.083
C04364=1141.540,66.995,-52.559,-179.642,6.507,149.083
C04365=1141.534,67.245,-52.575,-179.639,6.509,149.083
C04366=1141.530,67.494,-52.592,-179.636,6.509,149.082
C04367=1141.525,67.743,-52.608,-179.633,6.511,149.081
C04368=1141.520,67.992,-52.625,-179.631,6.513,149.081
C04369=1141.515,68.242,-52.640,-179.628,6.513,149.080
C04370=1141.510,68.491,-52.657,-179.625,6.515,149.080
C04371=1141.505,68.741,-52.674,-179.623,6.517,149.080
C04372=1141.501,68.990,-52.691,-179.620,6.517,149.079
C04373=1141.496,69.239,-52.707,-179.617,6.519,149.078
C04374=1141.490,69.490,-52.724,-179.614,6.520,149.078
C04375=1141.485,69.738,-52.740,-179.612,6.521,149.078
C04376=1141.480,69.988,-52.757,-179.609,6.522,149.077
C04377=1141.476,70.237,-52.773,-179.606,6.524,149.076
C04378=1141.470,70.486,-52.790,-179.604,6.525,149.076
C04379=1141.466,70.736,-52.807,-179.601,6.527,149.076
C04380=1141.461,70.985,-52.823,-179.598,6.528,149.075
C04381=1141.455,71.235,-52.840,-179.596,6.529,149.075
C04382=1141.451,71.485,-52.856,-179.593,6.530,149.074
C04383=1141.446,71.734,-52.873,-179.590,6.532,149.073
C04384=1141.440,71.983,-52.890,-179.588,6.533,149.073
C04385=1141.436,72.233,-52.907,-179.585,6.534,149.073
C04386=1141.431,72.481,-52.923,-179.582,6.536,149.072
C04387=1141.426,72.731,-52.940,-179.580,6.536,149.071
C04388=1141.421,72.981,-52.957,-179.577,6.538,149.071
C04389=1141.417,73.230,-52.973,-179.574,6.540,149.071
C04390=1141.411,73.479,-52.990,-179.572,6.541,149.070
C04391=1141.406,73.729,-53.007,-179.569,6.542,149.070
C04392=1141.401,73.979,-53.024,-179.566,6.543,149.069
C04393=1141.396,74.227,-53.041,-179.563,6.545,149.069
C04394=1141.392,74.477,-53.057,-179.561,6.546,149.068
C04395=1141.386,74.727,-53.075,-179.558,6.547,149.068
C04396=1141.381,74.975,-53.091,-179.555,6.549,149.067
C04397=1141.376,75.225,-53.108,-179.553,6.550,149.067
C04398=1141.372,75.475,-53.125,-179.550,6.551,149.066
C04399=1141.367,75.724,-53.141,-179.547,6.553,149.066
C04400=1141.361,75.973,-53.158,-179.544,6.554,149.065
C04401=1141.357,76.222,-53.176,-179.542,6.555,149.065
C04402=1141.352,76.472,-53.193,-179.539,6.557,149.064
C04403=1141.347,76.721,-53.210,-179.536,6.558,149.064
C04404=1141.342,76.971,-53.227,-179.534,6.559,149.063
C04405=1141.337,77.220,-53.243,-179.531,6.561,149.063
C04406=1141.332,77.470,-53.260,-179.528,6.562,149.062
C04407=1141.327,77.719,-53.277,-179.525,6.564,149.062
C04408=1141.322,77.968,-53.295,-179.523,6.565,149.061
C04409=1141.317,78.217,-53.311,-179.521,6.566,149.061
C04410=1141.312,78.467,-53.329,-179.517,6.567,149.060
C04411=1141.308,78.717,-53.345,-179.515,6.569,149.060
C04412=1141.302,78.966,-53.362,-179.512,6.570,149.059
C04413=1141.297,79.234,-53.380,-179.509,6.571,149.059
C04414=1141.292,79.503,-53.399,-179.506,6.573,149.058
C04415=1141.286,79.771,-53.418,-179.504,6.575,149.058
C04416=1141.281,80.039,-53.436,-179.501,6.576,149.057
C04417=1141.276,80.289,-53.453,-179.498,6.578,149.057
C04418=1141.272,80.538,-53.470,-179.495,6.579,149.056
C04419=1141.266,80.787,-53.488,-179.492,6.580,149.056
C04420=1141.261,81.037,-53.505,-179.490,6.581,149.055
C04421=1141.257,81.286,-53.522,-179.487,6.583,149.055
C04422=1141.251,81.536,-53.539,-179.484,6.585,149.054
C04423=1141.247,81.785,-53.556,-179.482,6.586,149.054
C04424=1141.242,82.035,-53.574,-179.479,6.587,149.053
C04425=1141.236,82.283,-53.591,-179.476,6.589,149.053
C04426=1141.232,82.533,-53.608,-179.473,6.590,149.052
C04427=1141.227,82.782,-53.625,-179.471,6.591,149.052
C04428=1141.222,83.032,-53.643,-179.468,6.592,149.051
C04429=1141.217,83.281,-53.660,-179.465,6.594,149.051
C04430=1141.212,83.531,-53.677,-179.462,6.596,149.051
C04431=1141.207,83.780,-53.695,-179.460,6.597,149.050
C04432=1141.202,84.029,-53.711,-179.457,6.598,149.049
C04433=1141.197,84.278,-53.729,-179.454,6.599,149.049
C04434=1141.192,84.528,-53.747,-179.452,6.601,149.049
C04435=1141.188,84.777,-53.764,-179.449,6.603,149.048
C04436=1141.183,85.026,-53.781,-179.447,6.604,149.048
C04437=1141.178,85.276,-53.799,-179.444,6.605,149.047
C04438=1141.173,85.525,-53.816,-179.441,6.607,149.047
C04439=1141.168,85.775,-53.833,-179.438,6.608,149.046
C04440=1141.163,86.024,-53.851,-179.436,6.609,149.046
C04441=1141.158,86.273,-53.869,-179.433,6.610,149.045
C04442=1141.154,86.523,-53.886,-179.430,6.612,149.045
C04443=1141.148,86.771,-53.903,-179.427,6.614,149.044
C04444=1141.143,87.021,-53.921,-179.424,6.615,149.044
C04445=1141.138,87.270,-53.939,-179.422,6.616,149.044
C04446=1141.134,87.520,-53.955,-179.419,6.618,149.043
C04447=1141.129,87.769,-53.973,-179.416,6.619,149.042
C04448=1141.123,88.019,-53.991,-179.414,6.621,149.042
C04449=1141.119,88.268,-54.009,-179.411,6.623,149.042
C04450=1141.114,88.517,-54.026,-179.409,6.624,149.041
C04451=1141.109,88.767,-54.043,-179.405,6.625,149.041
C04452=1141.104,89.016,-54.061,-179.403,6.626,149.040
C04453=1141.099,89.265,-54.079,-179.400,6.628,149.040
C04454=1141.094,89.515,-54.096,-179.397,6.630,149.039
C04455=1141.089,89.764,-54.114,-179.395,6.631,149.039
C04456=1141.084,90.013,-54.132,-179.392,6.632,149.038
C04457=1141.080,90.262,-54.149,-179.389,6.634,149.038
C04458=1141.075,90.512,-54.167,-179.386,6.635,149.037
C04459=1141.070,90.761,-54.185,-179.384,6.637,149.037
C04460=1141.065,91.011,-54.202,-179.381,6.639,149.036
C04461=1141.060,91.260,-54.220,-179.378,6.639,149.036
C04462=1141.055,91.509,-54.238,-179.376,6.641,149.035
C04463=1141.050,91.758,-54.256,-179.373,6.643,149.035
C04464=1141.045,92.008,-54.273,-179.370,6.644,149.035
C04465=1141.040,92.257,-54.291,-179.367,6.646,149.034
C04466=1141.036,92.506,-54.309,-179.364,6.647,149.034
C04467=1141.031,92.755,-54.327,-179.362,6.648,149.033
C04468=1141.026,93.005,-54.344,-179.359,6.650,149.033
C04469=1141.021,93.254,-54.362,-179.357,6.651,149.032
C04470=1141.016,93.504,-54.380,-179.354,6.653,149.032
C04471=1141.011,93.753,-54.398,-179.351,6.654,149.031
C04472=1141.007,94.002,-54.416,-179.348,6.656,149.031
C04473=1141.002,94.252,-54.434,-179.345,6.658,149.030
C04474=1140.996,94.501,-54.452,-179.343,6.659,149.030
C04475=1140.991,94.751,-54.470,-179.340,6.660,149.030
C04476=1140.987,95.000,-54.488,-179.337,6.662,149.029
C04477=1140.982,95.249,-54.506,-179.334,6.663,149.028
C04478=1140.977,95.498,-54.523,-179.332,6.665,149.028
C04479=1140.972,95.747,-54.541,-179.329,6.667,149.028
C04480=1140.967,95.996,-54.559,-179.326,6.668,149.027
C04481=1140.963,96.246,-54.578,-179.324,6.669,149.027
C04482=1140.958,96.495,-54.596,-179.321,6.670,149.026
C04483=1140.953,96.745,-54.614,-179.318,6.672,149.026
C04484=1140.948,96.994,-54.632,-179.315,6.674,149.025
C04485=1140.943,97.243,-54.650,-179.312,6.675,149.025
C04486=1140.938,97.492,-54.668,-179.310,6.677,149.024
C04487=1140.932,97.742,-54.686,-179.307,6.679,149.024
C04488=1140.927,97.991,-54.704,-179.304,6.680,149.023
C04489=1140.923,98.241,-54.723,-179.302,6.681,149.023
C04490=1140.918,98.490,-54.741,-179.299,6.683,149.023
C04491=1140.913,98.739,-54.759,-179.296,6.684,149.022
C04492=1140.908,98.988,-54.777,-179.293,6.686,149.022
C04493=1140.904,99.237,-54.795,-179.291,6.688,149.021
C04494=1140.899,99.487,-54.812,-179.288,6.689,149.021
C04495=1140.894,99.736,-54.831,-179.285,6.691,149.020
C04496=1140.889,99.986,-54.849,-179.282,6.692,149.020
C04497=1140.884,100.235,-54.867,-179.279,6.694,149.019
C04498=1140.879,100.484,-54.885,-179.277,6.695,149.019
C04499=1140.874,100.733,-54.904,-179.274,6.697,149.019
C04500=1140.870,100.983,-54.922,-179.272,6.698,149.018
C04501=1140.865,101.232,-54.940,-179.268,6.700,149.018
C04502=1140.859,101.481,-54.959,-179.266,6.701,149.017
C04503=1140.854,101.731,-54.977,-179.263,6.703,149.017
C04504=1140.850,101.980,-54.995,-179.260,6.705,149.016
C04505=1140.846,102.229,-55.014,-179.258,6.706,149.016
C04506=1140.841,102.478,-55.032,-179.255,6.708,149.015
C04507=1140.835,102.728,-55.051,-179.252,6.710,149.015
C04508=1140.830,102.977,-55.069,-179.249,6.710,149.014
C04509=1140.826,103.227,-55.087,-179.247,6.712,149.014
C04510=1140.821,103.475,-55.106,-179.244,6.713,149.014
C04511=1140.815,103.725,-55.124,-179.241,6.715,149.013
C04512=1140.811,103.974,-55.142,-179.239,6.717,149.013
C04513=1140.807,104.223,-55.161,-179.236,6.719,149.012
C04514=1140.802,104.472,-55.179,-179.233,6.720,149.012
C04515=1140.796,104.722,-55.198,-179.230,6.722,149.012
C04516=1140.792,104.972,-55.216,-179.227,6.723,149.011
C04517=1140.787,105.239,-55.236,-179.224,6.725,149.010
C04518=1140.781,105.508,-55.256,-179.222,6.727,149.010
C04519=1140.776,105.776,-55.276,-179.219,6.728,149.010
C04520=1140.770,106.045,-55.296,-179.215,6.730,149.009
C04521=1140.766,106.294,-55.315,-179.213,6.731,149.009
C04522=1140.761,106.543,-55.333,-179.210,6.733,149.008
C04523=1140.756,106.792,-55.352,-179.208,6.735,149.008
C04524=1140.752,107.042,-55.370,-179.205,6.736,149.007
C04525=1140.747,107.291,-55.388,-179.202,6.738,149.007
C04526=1140.741,107.540,-55.408,-179.199,6.740,149.007
C04527=1140.737,107.790,-55.426,-179.196,6.741,149.006
C04528=1140.732,108.039,-55.445,-179.193,6.743,149.006
C04529=1140.727,108.288,-55.463,-179.191,6.744,149.005
C04530=1140.723,108.537,-55.482,-179.188,6.746,149.005
C04531=1140.717,108.787,-55.501,-179.185,6.748,149.004
C04532=1140.713,109.035,-55.520,-179.182,6.749,149.004
C04533=1140.707,109.285,-55.538,-179.180,6.751,149.003
C04534=1140.703,109.534,-55.557,-179.177,6.753,149.003
C04535=1140.699,109.784,-55.576,-179.174,6.754,149.003
C04536=1140.693,110.033,-55.595,-179.172,6.756,149.002
C04537=1140.688,110.282,-55.613,-179.168,6.757,149.002
C04538=1140.684,110.531,-55.632,-179.166,6.759,149.001
C04539=1140.679,110.781,-55.650,-179.163,6.761,149.001
C04540=1140.673,111.029,-55.670,-179.160,6.762,149.000
C04541=1140.669,111.279,-55.689,-179.157,6.764,149.000
C04542=1140.664,111.528,-55.707,-179.155,6.766,149.000
C04543=1140.660,111.777,-55.726,-179.152,6.768,148.999
C04544=1140.654,112.027,-55.745,-179.149,6.769,148.999
C04545=1140.650,112.276,-55.764,-179.146,6.771,148.998
C04546=1140.645,112.525,-55.783,-179.144,6.773,148.998
C04547=1140.640,112.774,-55.801,-179.141,6.774,148.998
C04548=1140.635,113.024,-55.821,-179.138,6.776,148.997
C04549=1140.630,113.272,-55.840,-179.135,6.777,148.997
C04550=1140.625,113.523,-55.859,-179.132,6.779,148.996
C04551=1140.621,113.771,-55.877,-179.130,6.781,148.996
C04552=1140.616,114.021,-55.897,-179.127,6.782,148.995
C04553=1140.610,114.270,-55.916,-179.124,6.784,148.995
C04554=1140.606,114.519,-55.935,-179.121,6.786,148.994
C04555=1140.601,114.768,-55.954,-179.119,6.787,148.994
C04556=1140.597,115.018,-55.973,-179.116,6.789,148.994
C04557=1140.591,115.267,-55.992,-179.113,6.791,148.993
C04558=1140.586,115.516,-56.011,-179.111,6.792,148.993
C04559=1140.582,115.765,-56.030,-179.108,6.794,148.992
C04560=1140.577,116.014,-56.049,-179.105,6.796,148.992
C04561=1140.573,116.263,-56.068,-179.102,6.797,148.991
C04562=1140.567,116.512,-56.088,-179.099,6.799,148.991
C04563=1140.562,116.762,-56.106,-179.096,6.800,148.991
C04564=1140.558,117.011,-56.125,-179.094,6.802,148.990
C04565=1140.553,117.260,-56.145,-179.091,6.804,148.990
C04566=1140.548,117.510,-56.164,-179.088,6.806,148.989
C04567=1140.544,117.759,-56.183,-179.086,6.807,148.989
C04568=1140.539,118.008,-56.203,-179.083,6.809,148.989
C04569=1140.533,118.257,-56.222,-179.080,6.811,148.988
C04570=1140.529,118.507,-56.240,-179.077,6.812,148.988
C04571=1140.524,118.756,-56.260,-179.075,6.814,148.987
C04572=1140.519,119.005,-56.279,-179.072,6.816,148.987
C04573=1140.514,119.254,-56.299,-179.069,6.817,148.987
C04574=1140.510,119.503,-56.318,-179.066,6.819,148.986
C04575=1140.505,119.753,-56.337,-179.064,6.821,148.986
C04576=1140.500,120.002,-56.357,-179.061,6.822,148.985
C04577=1140.495,120.251,-56.376,-179.058,6.824,148.985
C04578=1140.490,120.500,-56.395,-179.056,6.826,148.985
C04579=1140.486,120.750,-56.415,-179.053,6.828,148.984
C04580=1140.480,120.998,-56.434,-179.050,6.829,148.984
C04581=1140.475,121.248,-56.454,-179.046,6.831,148.983
C04582=1140.471,121.497,-56.473,-179.044,6.833,148.983
C04583=1140.466,121.746,-56.492,-179.041,6.835,148.982
C04584=1140.461,121.996,-56.512,-179.038,6.836,148.982
C04585=1140.457,122.245,-56.532,-179.035,6.838,148.982
C04586=1140.452,122.494,-56.551,-179.033,6.840,148.981
C04587=1140.448,122.743,-56.570,-179.030,6.841,148.981
C04588=1140.442,122.992,-56.590,-179.027,6.843,148.980
C04589=1140.437,123.241,-56.609,-179.024,6.845,148.980
C04590=1140.433,123.491,-56.629,-179.022,6.847,148.980
C04591=1140.427,123.740,-56.648,-179.019,6.848,148.979
C04592=1140.423,123.989,-56.668,-179.016,6.850,148.979
C04593=1140.418,124.238,-56.688,-179.014,6.852,148.978
C04594=1140.414,124.487,-56.707,-179.011,6.853,148.978
C04595=1140.409,124.736,-56.727,-179.008,6.856,148.978
C04596=1140.404,124.986,-56.746,-179.005,6.858,148.977
C04597=1140.399,125.235,-56.766,-179.002,6.859,148.977
C04598=1140.394,125.484,-56.786,-178.999,6.861,148.976
C04599=1140.390,125.733,-56.806,-178.997,6.863,148.976
C04600=1140.385,125.983,-56.825,-178.994,6.864,148.976
C04601=1140.380,126.232,-56.845,-178.991,6.866,148.975
C04602=1140.375,126.481,-56.865,-178.988,6.868,148.975
C04603=1140.370,126.730,-56.885,-178.986,6.869,148.974
C04604=1140.365,126.979,-56.904,-178.983,6.871,148.974
C04605=1140.361,127.228,-56.924,-178.980,6.874,148.974
C04606=1140.357,127.477,-56.943,-178.977,6.875,148.973
C04607=1140.352,127.727,-56.963,-178.974,6.877,148.973
C04608=1140.347,127.975,-56.983,-178.972,6.879,148.972
C04609=1140.342,128.225,-57.003,-178.969,6.880,148.972
C04610=1140.337,128.474,-57.022,-178.966,6.882,148.972
C04611=1140.333,128.723,-57.043,-178.963,6.884,148.971
C04612=1140.327,128.972,-57.063,-178.961,6.885,148.971
C04613=1140.322,129.222,-57.082,-178.958,6.887,148.970
C04614=1140.318,129.471,-57.103,-178.955,6.890,148.970
C04615=1140.313,129.720,-57.122,-178.952,6.891,148.970
C04616=1140.308,129.969,-57.142,-178.949,6.893,148.969
C04617=1140.303,130.218,-57.162,-178.946,6.895,148.969
C04618=1140.299,130.467,-57.182,-178.944,6.896,148.968
C04619=1140.294,130.717,-57.202,-178.941,6.898,148.968
C04620=1140.289,130.966,-57.222,-178.938,6.900,148.968
C04621=1140.284,131.234,-57.243,-178.935,6.902,148.967
C04622=1140.278,131.503,-57.265,-178.932,6.904,148.967
C04623=1140.273,131.771,-57.286,-178.930,6.906,148.966
C04624=1140.268,132.040,-57.308,-178.926,6.908,148.966
C04625=1140.263,132.289,-57.328,-178.924,6.910,148.966
C04626=1140.259,132.538,-57.348,-178.921,6.912,148.965
C04627=1140.254,132.788,-57.368,-178.918,6.913,148.965
C04628=1140.250,133.037,-57.388,-178.915,6.915,148.964
C04629=1140.245,133.286,-57.409,-178.912,6.918,148.964
C04630=1140.239,133.535,-57.428,-178.909,6.919,148.964
C04631=1140.235,133.784,-57.449,-178.907,6.921,148.963
C04632=1140.230,134.033,-57.469,-178.904,6.923,148.963
C04633=1140.226,134.282,-57.489,-178.901,6.924,148.962
C04634=1140.221,134.531,-57.509,-178.898,6.926,148.962
C04635=1140.216,134.781,-57.530,-178.895,6.929,148.962
C04636=1140.211,135.030,-57.550,-178.892,6.930,148.961
C04637=1140.206,135.278,-57.570,-178.890,6.932,148.961
C04638=1140.201,135.528,-57.590,-178.887,6.934,148.961
C04639=1140.197,135.777,-57.610,-178.885,6.936,148.960
C04640=1140.192,136.026,-57.631,-178.882,6.937,148.960
C04641=1140.187,136.275,-57.651,-178.879,6.940,148.960
C04642=1140.183,136.525,-57.671,-178.876,6.942,148.959
C04643=1140.178,136.774,-57.691,-178.873,6.943,148.959
C04644=1140.173,137.023,-57.712,-178.871,6.945,148.958
C04645=1140.169,137.272,-57.733,-178.868,6.947,148.958
C04646=1140.164,137.521,-57.752,-178.865,6.948,148.958
C04647=1140.159,137.771,-57.773,-178.862,6.951,148.957
C04648=1140.154,138.020,-57.794,-178.859,6.953,148.957
C04649=1140.150,138.268,-57.814,-178.856,6.954,148.956
C04650=1140.145,138.517,-57.834,-178.854,6.956,148.956
C04651=1140.139,138.767,-57.854,-178.851,6.958,148.956
C04652=1140.135,139.016,-57.875,-178.848,6.960,148.955
C04653=1140.130,139.264,-57.895,-178.845,6.962,148.955
C04654=1140.125,139.514,-57.916,-178.843,6.964,148.955
C04655=1140.121,139.763,-57.936,-178.840,6.966,148.954
C04656=1140.116,140.012,-57.957,-178.837,6.967,148.954
C04657=1140.111,140.261,-57.978,-178.834,6.970,148.954
C04658=1140.107,140.510,-57.998,-178.831,6.972,148.953
C04659=1140.101,140.760,-58.018,-178.828,6.973,148.953
C04660=1140.097,141.009,-58.039,-178.826,6.975,148.952
C04661=1140.092,141.258,-58.059,-178.823,6.977,148.952
C04662=1140.087,141.507,-58.080,-178.820,6.979,148.952
C04663=1140.083,141.756,-58.100,-178.817,6.981,148.951
C04664=1140.078,142.005,-58.121,-178.815,6.983,148.951
C04665=1140.073,142.254,-58.142,-178.812,6.985,148.951
C04666=1140.069,142.503,-58.162,-178.809,6.987,148.950
C04667=1140.064,142.752,-58.183,-178.806,6.989,148.950
C04668=1140.059,143.001,-58.203,-178.803,6.991,148.950
C04669=1140.054,143.251,-58.225,-178.801,6.992,148.949
C04670=1140.050,143.499,-58.246,-178.798,6.994,148.949
C04671=1140.045,143.749,-58.267,-178.795,6.997,148.948
C04672=1140.041,143.998,-58.287,-178.792,6.998,148.948
C04673=1140.036,144.247,-58.308,-178.790,7.000,148.948
C04674=1140.031,144.496,-58.329,-178.787,7.002,148.947
C04675=1140.026,144.745,-58.349,-178.784,7.005,148.947
C04676=1140.022,144.994,-58.370,-178.781,7.006,148.947
C04677=1140.016,145.243,-58.391,-178.778,7.008,148.946
C04678=1140.012,145.492,-58.411,-178.775,7.010,148.946
C04679=1140.007,145.741,-58.433,-178.772,7.012,148.946
C04680=1140.003,145.990,-58.453,-178.769,7.014,148.945
C04681=1139.998,146.240,-58.475,-178.767,7.016,148.945
C04682=1139.993,146.489,-58.496,-178.764,7.018,148.945
C04683=1139.988,146.738,-58.516,-178.761,7.020,148.944
C04684=1139.984,146.987,-58.538,-178.758,7.022,148.944
C04685=1139.979,147.236,-58.558,-178.756,7.024,148.943
C04686=1139.974,147.485,-58.579,-178.753,7.025,148.943
C04687=1139.969,147.734,-58.600,-178.750,7.028,148.943
C04688=1139.965,147.983,-58.621,-178.747,7.030,148.943
C04689=1139.960,148.232,-58.642,-178.745,7.032,148.942
C04690=1139.956,148.481,-58.663,-178.741,7.034,148.942
C04691=1139.950,148.731,-58.684,-178.739,7.036,148.941
C04692=1139.946,148.979,-58.705,-178.736,7.038,148.941
C04693=1139.941,149.228,-58.726,-178.733,7.039,148.941
C04694=1139.936,149.478,-58.747,-178.730,7.042,148.940
C04695=1139.932,149.727,-58.769,-178.728,7.044,148.940
C04696=1139.927,149.976,-58.789,-178.725,7.046,148.940
C04697=1139.922,150.224,-58.811,-178.722,7.048,148.939
C04698=1139.917,150.474,-58.832,-178.719,7.050,148.939
C04699=1139.912,150.723,-58.853,-178.716,7.051,148.939
C04700=1139.908,150.971,-58.874,-178.714,7.053,148.938
C04701=1139.903,151.221,-58.895,-178.711,7.056,148.938
C04702=1139.898,151.470,-58.917,-178.708,7.058,148.938
C04703=1139.894,151.719,-58.937,-178.705,7.059,148.937
C04704=1139.889,151.968,-58.958,-178.702,7.062,148.937
C04705=1139.885,152.217,-58.980,-178.699,7.064,148.937
C04706=1139.879,152.467,-59.001,-178.697,7.066,148.936
C04707=1139.875,152.715,-59.023,-178.694,7.067,148.936
C04708=1139.870,152.964,-59.043,-178.691,7.070,148.936
C04709=1139.866,153.214,-59.065,-178.688,7.072,148.935
C04710=1139.861,153.463,-59.086,-178.686,7.073,148.935
C04711=1139.856,153.712,-59.108,-178.682,7.076,148.935
C04712=1139.851,153.960,-59.130,-178.680,7.078,148.934
C04713=1139.847,154.210,-59.150,-178.677,7.080,148.934
C04714=1139.842,154.458,-59.172,-178.674,7.082,148.934
C04715=1139.837,154.708,-59.193,-178.671,7.084,148.933
C04716=1139.832,154.956,-59.215,-178.669,7.086,148.933
C04717=1139.828,155.206,-59.237,-178.666,7.089,148.933
C04718=1139.823,155.455,-59.258,-178.663,7.090,148.932
C04719=1139.819,155.703,-59.279,-178.660,7.092,148.932
C04720=1139.814,155.953,-59.300,-178.657,7.094,148.932
C04721=1139.809,156.202,-59.322,-178.654,7.096,148.931
C04722=1139.804,156.451,-59.343,-178.652,7.098,148.931
C04723=1139.800,156.701,-59.365,-178.649,7.101,148.931
C04724=1139.795,156.949,-59.387,-178.646,7.103,148.930
C04725=1139.790,157.218,-59.409,-178.643,7.105,148.930
C04726=1139.785,157.487,-59.433,-178.640,7.107,148.930
C04727=1139.780,157.756,-59.456,-178.637,7.109,148.929
C04728=1139.775,158.025,-59.479,-178.634,7.111,148.929
C04729=1139.770,158.274,-59.501,-178.631,7.114,148.929
C04730=1139.765,158.523,-59.523,-178.629,7.116,148.928
C04731=1139.761,158.772,-59.545,-178.626,7.117,148.928
C04732=1139.756,159.021,-59.567,-178.623,7.120,148.928
C04733=1139.751,159.270,-59.588,-178.620,7.122,148.927
C04734=1139.746,159.519,-59.610,-178.617,7.124,148.927
C04735=1139.742,159.768,-59.631,-178.614,7.126,148.927
C04736=1139.737,160.017,-59.653,-178.612,7.128,148.926
C04737=1139.732,160.266,-59.675,-178.608,7.130,148.926
C04738=1139.728,160.514,-59.697,-178.606,7.132,148.926
C04739=1139.723,160.764,-59.718,-178.603,7.134,148.925
C04740=1139.718,161.013,-59.740,-178.600,7.137,148.925
C04741=1139.714,161.262,-59.762,-178.597,7.138,148.925
C04742=1139.709,161.511,-59.783,-178.595,7.141,148.925
C04743=1139.705,161.760,-59.805,-178.592,7.143,148.924
C04744=1139.700,162.009,-59.827,-178.589,7.145,148.924
C04745=1139.695,162.258,-59.849,-178.586,7.147,148.923
C04746=1139.691,162.507,-59.871,-178.584,7.149,148.923
C04747=1139.686,162.756,-59.893,-178.581,7.151,148.923
C04748=1139.682,163.005,-59.915,-178.578,7.154,148.922
C04749=1139.677,163.254,-59.936,-178.575,7.156,148.922
C04750=1139.672,163.503,-59.959,-178.572,7.158,148.922
C04751=1139.667,163.752,-59.981,-178.569,7.160,148.922
C04752=1139.662,164.001,-60.003,-178.567,7.162,148.921
C04753=1139.658,164.250,-60.024,-178.564,7.164,148.921
C04754=1139.653,164.499,-60.046,-178.561,7.166,148.921
C04755=1139.648,164.748,-60.068,-178.558,7.169,148.920
C04756=1139.644,164.997,-60.090,-178.555,7.170,148.920
C04757=1139.639,165.246,-60.112,-178.553,7.173,148.920
C04758=1139.635,165.495,-60.135,-178.550,7.175,148.919
C04759=1139.630,165.744,-60.157,-178.547,7.177,148.919
C04760=1139.626,165.993,-60.179,-178.544,7.180,148.919
C04761=1139.621,166.242,-60.201,-178.541,7.181,148.919
C04762=1139.616,166.491,-60.223,-178.539,7.183,148.918
C04763=1139.611,166.740,-60.245,-178.535,7.186,148.918
C04764=1139.607,166.989,-60.267,-178.533,7.188,148.918
C04765=1139.602,167.237,-60.289,-178.530,7.190,148.917
C04766=1139.597,167.487,-60.312,-178.527,7.192,148.917
C04767=1139.592,167.735,-60.334,-178.524,7.195,148.917
C04768=1139.588,167.985,-60.356,-178.522,7.197,148.916
C04769=1139.584,168.234,-60.378,-178.519,7.198,148.916
C04770=1139.578,168.482,-60.401,-178.516,7.201,148.916
C04771=1139.574,168.732,-60.423,-178.513,7.203,148.916
C04772=1139.569,168.980,-60.445,-178.510,7.205,148.915
C04773=1139.564,169.230,-60.468,-178.508,7.207,148.915
C04774=1139.560,169.478,-60.490,-178.505,7.210,148.915
C04775=1139.555,169.727,-60.512,-178.502,7.212,148.914
C04776=1139.551,169.977,-60.535,-178.499,7.213,148.914
C04777=1139.546,170.225,-60.557,-178.496,7.216,148.914
C04778=1139.541,170.474,-60.579,-178.494,7.218,148.913
C04779=1139.536,170.723,-60.602,-178.490,7.221,148.913
C04780=1139.532,170.972,-60.624,-178.488,7.223,148.913
C04781=1139.528,171.222,-60.646,-178.485,7.225,148.913
C04782=1139.522,171.470,-60.669,-178.482,7.227,148.912
C04783=1139.518,171.719,-60.691,-178.479,7.230,148.912
C04784=1139.513,171.968,-60.714,-178.477,7.232,148.912
C04785=1139.508,172.217,-60.736,-178.473,7.234,148.911
C04786=1139.504,172.466,-60.759,-178.471,7.236,148.911
C04787=1139.499,172.715,-60.781,-178.468,7.238,148.911
C04788=1139.495,172.963,-60.804,-178.466,7.241,148.911
C04789=1139.490,173.213,-60.826,-178.463,7.242,148.910
C04790=1139.485,173.461,-60.849,-178.460,7.245,148.910
C04791=1139.480,173.711,-60.871,-178.457,7.247,148.910
C04792=1139.476,173.959,-60.894,-178.454,7.250,148.910
C04793=1139.472,174.209,-60.916,-178.451,7.251,148.909
C04794=1139.467,174.457,-60.939,-178.449,7.254,148.909
C04795=1139.463,174.706,-60.961,-178.446,7.256,148.909
C04796=1139.458,174.955,-60.985,-178.443,7.258,148.908
C04797=1139.453,175.204,-61.006,-178.440,7.261,148.908
C04798=1139.448,175.453,-61.030,-178.437,7.263,148.908
C04799=1139.444,175.702,-61.052,-178.434,7.265,148.907
C04800=1139.439,175.951,-61.075,-178.432,7.268,148.907
C04801=1139.434,176.200,-61.098,-178.429,7.269,148.907
C04802=1139.430,176.448,-61.121,-178.426,7.272,148.907
C04803=1139.425,176.698,-61.143,-178.423,7.274,148.906
C04804=1139.420,176.946,-61.166,-178.420,7.277,148.906
C04805=1139.416,177.195,-61.189,-178.418,7.279,148.906
C04806=1139.412,177.444,-61.211,-178.415,7.281,148.906
C04807=1139.407,177.694,-61.235,-178.412,7.283,148.905
C04808=1139.402,177.942,-61.257,-178.409,7.286,148.905
C04809=1139.397,178.191,-61.280,-178.406,7.288,148.905
C04810=1139.393,178.440,-61.303,-178.403,7.290,148.905
C04811=1139.389,178.689,-61.326,-178.401,7.292,148.904
C04812=1139.384,178.938,-61.349,-178.398,7.295,148.904
C04813=1139.378,179.187,-61.371,-178.395,7.297,148.904
C04814=1139.374,179.436,-61.394,-178.392,7.299,148.903
C04815=1139.370,179.685,-61.417,-178.390,7.301,148.903
C04816=1139.366,179.933,-61.440,-178.386,7.304,148.903
C04817=1139.361,180.182,-61.464,-178.384,7.306,148.903
C04818=1139.356,180.431,-61.487,-178.381,7.309,148.902
C04819=1139.351,180.680,-61.509,-178.378,7.310,148.902
C04820=1139.347,180.929,-61.532,-178.375,7.313,148.902
C04821=1139.342,181.178,-61.555,-178.372,7.316,148.902
C04822=1139.337,181.427,-61.579,-178.370,7.318,148.901
C04823=1139.333,181.676,-61.601,-178.367,7.320,148.901
C04824=1139.329,181.925,-61.625,-178.364,7.322,148.901
C04825=1139.323,182.173,-61.648,-178.361,7.325,148.901
C04826=1139.319,182.422,-61.671,-178.358,7.327,148.900
C04827=1139.315,182.671,-61.694,-178.356,7.330,148.900
C04828=1139.310,182.920,-61.717,-178.353,7.331,148.900
C04829=1139.305,183.190,-61.742,-178.350,7.334,148.900
C04830=1139.300,183.459,-61.767,-178.347,7.337,148.899
C04831=1139.295,183.728,-61.793,-178.343,7.339,148.899
C04832=1139.290,183.999,-61.818,-178.340,7.342,148.899
C04833=1139.286,184.248,-61.841,-178.338,7.344,148.899
C04834=1139.280,184.496,-61.864,-178.335,7.346,148.898
C04835=1139.276,184.745,-61.887,-178.332,7.348,148.898
C04836=1139.272,184.994,-61.910,-178.329,7.351,148.898
C04837=1139.267,185.243,-61.934,-178.326,7.354,148.898
C04838=1139.262,185.492,-61.957,-178.324,7.356,148.897
C04839=1139.258,185.741,-61.981,-178.321,7.359,148.897
C04840=1139.253,185.990,-62.004,-178.318,7.360,148.897
C04841=1139.248,186.239,-62.028,-178.315,7.363,148.897
C04842=1139.245,186.487,-62.051,-178.313,7.365,148.896
C04843=1139.240,186.736,-62.074,-178.310,7.368,148.896
C04844=1139.235,186.985,-62.097,-178.307,7.370,148.896
C04845=1139.230,187.234,-62.121,-178.304,7.372,148.895
C04846=1139.226,187.483,-62.144,-178.301,7.375,148.895
C04847=1139.221,187.732,-62.168,-178.298,7.377,148.895
C04848=1139.217,187.981,-62.192,-178.296,7.380,148.895
C04849=1139.212,188.230,-62.215,-178.293,7.381,148.894
C04850=1139.207,188.479,-62.238,-178.290,7.384,148.894
C04851=1139.203,188.727,-62.262,-178.287,7.387,148.894
C04852=1139.198,188.976,-62.286,-178.284,7.389,148.894
C04853=1139.193,189.225,-62.309,-178.281,7.391,148.894
C04854=1139.189,189.474,-62.333,-178.279,7.393,148.893
C04855=1139.184,189.723,-62.357,-178.276,7.396,148.893
C04856=1139.180,189.972,-62.380,-178.273,7.399,148.893
C04857=1139.175,190.220,-62.404,-178.270,7.401,148.893
C04858=1139.171,190.469,-62.427,-178.267,7.404,148.892
C04859=1139.166,190.718,-62.451,-178.265,7.405,148.892
C04860=1139.161,190.967,-62.475,-178.262,7.408,148.892
C04861=1139.157,191.216,-62.498,-178.259,7.411,148.892
C04862=1139.152,191.465,-62.521,-178.256,7.413,148.892
C04863=1139.148,191.713,-62.546,-178.253,7.415,148.891
C04864=1139.143,191.962,-62.569,-178.250,7.418,148.891
C04865=1139.139,192.211,-62.593,-178.248,7.420,148.891
C04866=1139.134,192.460,-62.616,-178.245,7.423,148.891
C04867=1139.129,192.708,-62.640,-178.243,7.425,148.890
C04868=1139.125,192.957,-62.664,-178.239,7.427,148.890
C04869=1139.120,193.206,-62.688,-178.236,7.430,148.890
C04870=1139.115,193.455,-62.712,-178.234,7.432,148.890
C04871=1139.111,193.704,-62.736,-178.231,7.435,148.890
C04872=1139.106,193.953,-62.760,-178.228,7.438,148.889
C04873=1139.102,194.201,-62.784,-178.225,7.440,148.889
C04874=1139.097,194.451,-62.807,-178.222,7.442,148.889
C04875=1139.093,194.699,-62.831,-178.219,7.445,148.889
C04876=1139.088,194.948,-62.854,-178.217,7.447,148.888
C04877=1139.083,195.197,-62.879,-178.214,7.450,148.888
C04878=1139.079,195.445,-62.903,-178.212,7.452,148.888
C04879=1139.075,195.695,-62.927,-178.208,7.454,148.888
C04880=1139.070,195.943,-62.951,-178.205,7.457,148.888
C04881=1139.066,196.192,-62.975,-178.203,7.459,148.887
C04882=1139.060,196.441,-62.999,-178.200,7.462,148.887
C04883=1139.056,196.689,-63.023,-178.197,7.464,148.887
C04884=1139.052,196.938,-63.047,-178.194,7.466,148.887
C04885=1139.048,197.188,-63.071,-178.192,7.469,148.887
C04886=1139.042,197.436,-63.096,-178.188,7.472,148.886
C04887=1139.038,197.685,-63.120,-178.186,7.474,148.886
C04888=1139.033,197.934,-63.143,-178.183,7.477,148.886
C04889=1139.029,198.182,-63.167,-178.180,7.479,148.886
C04890=1139.024,198.432,-63.192,-178.177,7.481,148.885
C04891=1139.020,198.680,-63.216,-178.175,7.484,148.885
C04892=1139.016,198.928,-63.240,-178.172,7.487,148.885
C04893=1139.010,199.178,-63.264,-178.169,7.489,148.885
C04894=1139.006,199.426,-63.288,-178.166,7.492,148.885
C04895=1139.002,199.675,-63.313,-178.163,7.494,148.884
C04896=1138.997,199.924,-63.337,-178.161,7.496,148.884
C04897=1138.992,200.172,-63.361,-178.158,7.499,148.884
C04898=1138.988,200.421,-63.386,-178.155,7.502,148.884
C04899=1138.983,200.671,-63.410,-178.152,7.505,148.884
C04900=1138.979,200.919,-63.434,-178.149,7.506,148.883
C04901=1138.974,201.168,-63.458,-178.146,7.509,148.883
C04902=1138.969,201.416,-63.483,-178.144,7.512,148.883
C04903=1138.965,201.666,-63.507,-178.141,7.514,148.883
C04904=1138.961,201.914,-63.531,-178.138,7.517,148.883
C04905=1138.956,202.163,-63.556,-178.135,7.520,148.882
C04906=1138.952,202.412,-63.580,-178.133,7.521,148.882
C04907=1138.947,202.660,-63.605,-178.130,7.524,148.882
C04908=1138.943,202.909,-63.629,-178.126,7.527,148.882
C04909=1138.938,203.158,-63.654,-178.124,7.530,148.882
C04910=1138.934,203.407,-63.678,-178.121,7.532,148.881
C04911=1138.929,203.655,-63.702,-178.118,7.534,148.881
C04912=1138.924,203.904,-63.727,-178.115,7.537,148.881
C04913=1138.920,204.153,-63.751,-178.113,7.539,148.881
C04914=1138.915,204.402,-63.776,-178.110,7.542,148.881
C04915=1138.911,204.650,-63.800,-178.107,7.545,148.880
C04916=1138.906,204.900,-63.825,-178.104,7.548,148.880
C04917=1138.902,205.148,-63.849,-178.102,7.549,148.880
C04918=1138.897,205.396,-63.875,-178.099,7.552,148.880
C04919=1138.893,205.645,-63.900,-178.096,7.555,148.880
C04920=1138.888,205.894,-63.924,-178.093,7.558,148.879
C04921=1138.884,206.143,-63.949,-178.090,7.560,148.879
C04922=1138.879,206.392,-63.973,-178.088,7.563,148.879
C04923=1138.874,206.640,-63.997,-178.084,7.565,148.879
C04924=1138.871,206.889,-64.023,-178.082,7.567,148.879
C04925=1138.866,207.138,-64.047,-178.079,7.570,148.879
C04926=1138.860,207.386,-64.072,-178.076,7.573,148.878
C04927=1138.857,207.636,-64.096,-178.073,7.576,148.878
C04928=1138.852,207.884,-64.122,-178.071,7.578,148.878
C04929=1138.848,208.133,-64.146,-178.068,7.580,148.878
C04930=1138.843,208.381,-64.171,-178.065,7.583,148.878
C04931=1138.838,208.631,-64.196,-178.062,7.586,148.878
C04932=1138.834,208.879,-64.221,-178.059,7.588,148.877
C04933=1138.830,209.150,-64.248,-178.056,7.592,148.877
C04934=1138.824,209.420,-64.275,-178.053,7.595,148.877
C04935=1138.819,209.691,-64.302,-178.050,7.597,148.877
C04936=1138.814,209.961,-64.329,-178.047,7.600,148.877
C04937=1138.810,210.211,-64.354,-178.044,7.603,148.876
C04938=1138.805,210.458,-64.379,-178.042,7.605,148.876
C04939=1138.801,210.708,-64.404,-178.039,7.608,148.876
C04940=1138.796,210.956,-64.428,-178.036,7.611,148.876
C04941=1138.792,211.205,-64.454,-178.033,7.613,148.876
C04942=1138.787,211.454,-64.478,-178.030,7.615,148.875
C04943=1138.783,211.702,-64.504,-178.028,7.618,148.875
C04944=1138.778,211.951,-64.529,-178.024,7.621,148.875
C04945=1138.774,212.200,-64.554,-178.022,7.624,148.875
C04946=1138.769,212.448,-64.579,-178.019,7.626,148.875
C04947=1138.765,212.697,-64.604,-178.017,7.629,148.875
C04948=1138.760,212.946,-64.629,-178.013,7.631,148.874
C04949=1138.756,213.195,-64.655,-178.010,7.634,148.874
C04950=1138.751,213.443,-64.679,-178.008,7.637,148.874
C04951=1138.747,213.692,-64.705,-178.005,7.640,148.874
C04952=1138.742,213.941,-64.729,-178.002,7.642,148.874
C04953=1138.738,214.189,-64.755,-177.999,7.644,148.874
C04954=1138.733,214.438,-64.780,-177.997,7.647,148.874
C04955=1138.728,214.687,-64.805,-177.994,7.650,148.873
C04956=1138.725,214.936,-64.831,-177.990,7.653,148.873
C04957=1138.720,215.184,-64.855,-177.988,7.655,148.873
C04958=1138.715,215.433,-64.881,-177.985,7.658,148.873
C04959=1138.711,215.681,-64.906,-177.983,7.661,148.873
C04960=1138.706,215.931,-64.931,-177.979,7.663,148.873
C04961=1138.701,216.179,-64.957,-177.977,7.666,148.872
C04962=1138.697,216.427,-64.982,-177.974,7.668,148.872
C04963=1138.693,216.676,-65.008,-177.972,7.671,148.872
C04964=1138.688,216.925,-65.032,-177.969,7.674,148.872
C04965=1138.684,217.173,-65.058,-177.965,7.677,148.872
C04966=1138.680,217.422,-65.084,-177.963,7.680,148.872
C04967=1138.675,217.670,-65.109,-177.960,7.682,148.872
C04968=1138.671,217.920,-65.134,-177.958,7.685,148.871
C04969=1138.666,218.168,-65.160,-177.954,7.687,148.871
C04970=1138.662,218.417,-65.185,-177.952,7.690,148.871
C04971=1138.657,218.666,-65.211,-177.949,7.693,148.871
C04972=1138.653,218.914,-65.236,-177.946,7.696,148.871
C04973=1138.648,219.163,-65.262,-177.943,7.699,148.871
C04974=1138.644,219.412,-65.287,-177.940,7.700,148.870
C04975=1138.639,219.660,-65.313,-177.938,7.703,148.870
C04976=1138.635,219.909,-65.338,-177.935,7.706,148.870
C04977=1138.630,220.158,-65.364,-177.932,7.709,148.870
C04978=1138.626,220.406,-65.390,-177.929,7.712,148.870
C04979=1138.621,220.654,-65.415,-177.926,7.715,148.870
C04980=1138.617,220.903,-65.441,-177.923,7.718,148.870
C04981=1138.612,221.151,-65.466,-177.921,7.720,148.870
C04982=1138.608,221.400,-65.492,-177.918,7.723,148.869
C04983=1138.603,221.649,-65.519,-177.915,7.725,148.869
C04984=1138.599,221.898,-65.544,-177.913,7.728,148.869
C04985=1138.594,222.146,-65.570,-177.909,7.731,148.869
C04986=1138.590,222.395,-65.595,-177.906,7.734,148.869
C04987=1138.586,222.644,-65.621,-177.904,7.737,148.869
C04988=1138.581,222.892,-65.647,-177.901,7.739,148.869
C04989=1138.577,223.141,-65.672,-177.899,7.742,148.869
C04990=1138.572,223.390,-65.698,-177.896,7.745,148.868
C04991=1138.567,223.639,-65.724,-177.893,7.748,148.868
C04992=1138.563,223.887,-65.750,-177.890,7.750,148.868
C04993=1138.558,224.136,-65.776,-177.887,7.753,148.868
C04994=1138.554,224.384,-65.801,-177.884,7.756,148.868
C04995=1138.550,224.633,-65.828,-177.881,7.759,148.868
C04996=1138.546,224.881,-65.854,-177.879,7.761,148.868
C04997=1138.540,225.130,-65.879,-177.876,7.764,148.868
C04998=1138.536,225.379,-65.905,-177.873,7.767,148.867
C04999=1138.532,225.627,-65.931,-177.870,7.769,148.867
C05000=1138.528,225.876,-65.957,-177.867,7.772,148.867
C05001=1138.523,226.125,-65.984,-177.865,7.775,148.867
C05002=1138.518,226.373,-66.009,-177.862,7.778,148.867
C05003=1138.514,226.622,-66.035,-177.859,7.781,148.867
C05004=1138.510,226.870,-66.061,-177.857,7.783,148.867
C05005=1138.505,227.119,-66.088,-177.854,7.786,148.867
C05006=1138.501,227.368,-66.114,-177.851,7.789,148.866
C05007=1138.496,227.616,-66.139,-177.848,7.791,148.866
C05008=1138.491,227.864,-66.166,-177.845,7.794,148.866
C05009=1138.487,228.113,-66.192,-177.842,7.797,148.866
C05010=1138.483,228.362,-66.217,-177.840,7.800,148.866
C05011=1138.478,228.610,-66.245,-177.837,7.803,148.866
C05012=1138.474,228.859,-66.270,-177.834,7.806,148.866
C05013=1138.470,229.108,-66.296,-177.831,7.809,148.866
C05014=1138.465,229.357,-66.323,-177.828,7.812,148.866
C05015=1138.460,229.605,-66.348,-177.826,7.814,148.865
C05016=1138.457,229.853,-66.375,-177.823,7.817,148.865
C05017=1138.452,230.102,-66.401,-177.820,7.819,148.865
C05018=1138.447,230.351,-66.427,-177.817,7.822,148.865
C05019=1138.443,230.599,-66.453,-177.814,7.825,148.865
C05020=1138.438,230.848,-66.480,-177.812,7.828,148.865
C05021=1138.435,231.096,-66.506,-177.809,7.831,148.865
C05022=1138.430,231.345,-66.533,-177.806,7.834,148.865
C05023=1138.426,231.594,-66.559,-177.803,7.837,148.865
C05024=1138.421,231.843,-66.585,-177.800,7.840,148.864
C05025=1138.417,232.091,-66.612,-177.798,7.843,148.864
C05026=1138.412,232.339,-66.639,-177.795,7.846,148.864
C05027=1138.407,232.587,-66.664,-177.792,7.848,148.864
C05028=1138.403,232.836,-66.691,-177.789,7.851,148.864
C05029=1138.398,233.085,-66.717,-177.787,7.853,148.864
C05030=1138.394,233.333,-66.744,-177.784,7.856,148.864
C05031=1138.390,233.581,-66.771,-177.781,7.859,148.864
C05032=1138.385,233.831,-66.797,-177.778,7.862,148.864
C05033=1138.381,234.079,-66.824,-177.775,7.865,148.863
C05034=1138.376,234.328,-66.850,-177.772,7.868,148.863
C05035=1138.372,234.576,-66.876,-177.770,7.871,148.863
C05036=1138.367,234.824,-66.903,-177.767,7.873,148.863
C05037=1138.364,235.096,-66.933,-177.764,7.876,148.863
C05038=1138.358,235.369,-66.961,-177.761,7.880,148.863
C05039=1138.353,235.640,-66.991,-177.758,7.883,148.863
C05040=1138.349,235.913,-67.020,-177.755,7.886,148.863
C05041=1138.344,236.161,-67.046,-177.752,7.889,148.863
C05042=1138.340,236.410,-67.073,-177.749,7.892,148.863
C05043=1138.336,236.658,-67.100,-177.747,7.895,148.863
C05044=1138.331,236.907,-67.127,-177.744,7.898,148.863
C05045=1138.326,237.155,-67.154,-177.741,7.900,148.862
C05046=1138.322,237.404,-67.179,-177.738,7.903,148.862
C05047=1138.318,237.652,-67.206,-177.735,7.906,148.862
C05048=1138.313,237.901,-67.234,-177.733,7.909,148.862
C05049=1138.309,238.149,-67.260,-177.730,7.912,148.862
C05050=1138.304,238.398,-67.287,-177.727,7.915,148.862
C05051=1138.300,238.646,-67.314,-177.724,7.918,148.862
C05052=1138.296,238.894,-67.341,-177.721,7.921,148.862
C05053=1138.291,239.143,-67.368,-177.719,7.924,148.862
C05054=1138.286,239.391,-67.395,-177.716,7.927,148.862
C05055=1138.282,239.640,-67.422,-177.713,7.930,148.862
C05056=1138.278,239.889,-67.449,-177.710,7.932,148.862
C05057=1138.274,240.137,-67.476,-177.707,7.935,148.861
C05058=1138.269,240.386,-67.503,-177.705,7.938,148.861
C05059=1138.264,240.634,-67.530,-177.702,7.941,148.861
C05060=1138.261,240.882,-67.556,-177.699,7.944,148.861
C05061=1138.256,241.131,-67.583,-177.696,7.947,148.861
C05062=1138.251,241.379,-67.610,-177.693,7.950,148.861
C05063=1138.247,241.628,-67.638,-177.691,7.953,148.861
C05064=1138.243,241.877,-67.665,-177.688,7.956,148.861
C05065=1138.239,242.125,-67.691,-177.685,7.959,148.861
C05066=1138.234,242.374,-67.718,-177.682,7.962,148.861
C05067=1138.229,242.622,-67.745,-177.679,7.965,148.861
C05068=1138.225,242.871,-67.772,-177.677,7.967,148.861
C05069=1138.221,243.120,-67.800,-177.674,7.970,148.861
C05070=1138.217,243.367,-67.827,-177.671,7.973,148.860
C05071=1138.212,243.616,-67.854,-177.668,7.976,148.860
C05072=1138.208,243.864,-67.881,-177.665,7.979,148.860
C05073=1138.203,244.113,-67.908,-177.663,7.982,148.860
C05074=1138.199,244.362,-67.936,-177.660,7.985,148.860
C05075=1138.195,244.610,-67.963,-177.657,7.988,148.860
C05076=1138.190,244.858,-67.991,-177.654,7.991,148.860
C05077=1138.185,245.107,-68.018,-177.651,7.994,148.860
C05078=1138.181,245.355,-68.045,-177.649,7.997,148.860
C05079=1138.177,245.604,-68.073,-177.646,7.999,148.860
C05080=1138.172,245.853,-68.100,-177.643,8.002,148.860
C05081=1138.168,246.101,-68.126,-177.640,8.005,148.860
C05082=1138.164,246.349,-68.153,-177.638,8.009,148.860
C05083=1138.160,246.598,-68.182,-177.635,8.011,148.860
C05084=1138.155,246.846,-68.209,-177.632,8.014,148.860
C05085=1138.151,247.094,-68.236,-177.630,8.017,148.860
C05086=1138.146,247.343,-68.263,-177.627,8.020,148.859
C05087=1138.142,247.592,-68.291,-177.624,8.023,148.859
C05088=1138.138,247.840,-68.319,-177.621,8.026,148.859
C05089=1138.133,248.088,-68.346,-177.618,8.029,148.859
C05090=1138.129,248.337,-68.374,-177.615,8.033,148.859
C05091=1138.124,248.586,-68.402,-177.612,8.036,148.859
C05092=1138.119,248.834,-68.429,-177.609,8.039,148.859
C05093=1138.116,249.083,-68.457,-177.607,8.041,148.859
C05094=1138.111,249.331,-68.484,-177.604,8.045,148.859
C05095=1138.107,249.579,-68.512,-177.601,8.048,148.859
C05096=1138.103,249.828,-68.539,-177.599,8.050,148.859
C05097=1138.098,250.076,-68.567,-177.596,8.053,148.859
C05098=1138.094,250.325,-68.594,-177.593,8.056,148.859
C05099=1138.090,250.573,-68.622,-177.590,8.059,148.859
C05100=1138.085,250.821,-68.650,-177.587,8.062,148.859
C05101=1138.081,251.070,-68.677,-177.585,8.065,148.859
C05102=1138.076,251.318,-68.706,-177.582,8.068,148.859
C05103=1138.072,251.567,-68.733,-177.579,8.071,148.859
C05104=1138.067,251.815,-68.760,-177.577,8.074,148.859
C05105=1138.064,252.063,-68.789,-177.574,8.077,148.859
C05106=1138.059,252.312,-68.816,-177.571,8.080,148.858
C05107=1138.055,252.560,-68.844,-177.568,8.084,148.858
C05108=1138.050,252.809,-68.872,-177.565,8.087,148.858
C05109=1138.045,253.057,-68.899,-177.562,8.090,148.858
C05110=1138.042,253.306,-68.927,-177.559,8.092,148.858
C05111=1138.037,253.554,-68.955,-177.557,8.096,148.858
C05112=1138.034,253.802,-68.983,-177.554,8.099,148.858
C05113=1138.028,254.051,-69.011,-177.551,8.102,148.858
C05114=1138.024,254.299,-69.039,-177.549,8.104,148.858
C05115=1138.020,254.547,-69.067,-177.546,8.107,148.858
C05116=1138.016,254.795,-69.095,-177.543,8.110,148.858
C05117=1138.011,255.045,-69.123,-177.540,8.113,148.858
C05118=1138.007,255.293,-69.150,-177.538,8.116,148.858
C05119=1138.003,255.541,-69.179,-177.534,8.120,148.858
C05120=1137.998,255.789,-69.207,-177.532,8.123,148.858
C05121=1137.994,256.038,-69.235,-177.529,8.126,148.858
C05122=1137.990,256.286,-69.263,-177.526,8.129,148.858
C05123=1137.985,256.535,-69.292,-177.523,8.132,148.858
C05124=1137.980,256.783,-69.319,-177.521,8.135,148.858
C05125=1137.976,257.031,-69.346,-177.518,8.138,148.858
C05126=1137.972,257.280,-69.375,-177.515,8.141,148.858
C05127=1137.967,257.528,-69.403,-177.513,8.144,148.858
C05128=1137.964,257.776,-69.431,-177.510,8.147,148.858
C05129=1137.959,258.025,-69.460,-177.507,8.151,148.858
C05130=1137.955,258.273,-69.488,-177.504,8.154,148.858
C05131=1137.951,258.522,-69.516,-177.501,8.157,148.858
C05132=1137.946,258.770,-69.544,-177.498,8.160,148.858
C05133=1137.942,259.019,-69.572,-177.496,8.163,148.858
C05134=1137.937,259.267,-69.601,-177.493,8.165,148.857
C05135=1137.933,259.515,-69.629,-177.490,8.169,148.858
C05136=1137.928,259.764,-69.657,-177.488,8.172,148.858
C05137=1137.924,260.012,-69.685,-177.485,8.175,148.857
C05138=1137.919,260.260,-69.714,-177.482,8.178,148.857
C05139=1137.916,260.508,-69.742,-177.479,8.181,148.857
C05140=1137.912,260.757,-69.771,-177.476,8.184,148.858
C05141=1137.907,261.030,-69.802,-177.474,8.187,148.857
C05142=1137.902,261.304,-69.833,-177.470,8.191,148.857
C05143=1137.897,261.578,-69.864,-177.467,8.194,148.857
C05144=1137.893,261.851,-69.896,-177.464,8.198,148.857
C05145=1137.888,262.100,-69.924,-177.462,8.201,148.858
C05146=1137.883,262.348,-69.953,-177.459,8.204,148.857
C05147=1137.880,262.597,-69.981,-177.456,8.207,148.857
C05148=1137.875,262.844,-70.010,-177.453,8.211,148.857
C05149=1137.871,263.093,-70.038,-177.450,8.213,148.857
C05150=1137.867,263.342,-70.067,-177.448,8.217,148.857
C05151=1137.862,263.589,-70.095,-177.445,8.220,148.857
C05152=1137.858,263.838,-70.124,-177.442,8.223,148.857
C05153=1137.854,264.087,-70.153,-177.439,8.225,148.857
C05154=1137.849,264.334,-70.181,-177.437,8.229,148.857
C05155=1137.845,264.583,-70.210,-177.433,8.232,148.857
C05156=1137.840,264.831,-70.238,-177.431,8.235,148.857
C05157=1137.836,265.080,-70.267,-177.428,8.238,148.857
C05158=1137.832,265.328,-70.296,-177.426,8.242,148.857
C05159=1137.828,265.576,-70.324,-177.423,8.244,148.857
C05160=1137.823,265.824,-70.353,-177.420,8.247,148.857
C05161=1137.819,266.073,-70.382,-177.417,8.251,148.857
C05162=1137.815,266.322,-70.411,-177.414,8.254,148.857
C05163=1137.810,266.569,-70.439,-177.411,8.257,148.857
C05164=1137.806,266.818,-70.468,-177.409,8.260,148.857
C05165=1137.802,267.066,-70.497,-177.406,8.263,148.857
C05166=1137.797,267.314,-70.525,-177.403,8.266,148.857
C05167=1137.793,267.562,-70.555,-177.400,8.270,148.857
C05168=1137.789,267.811,-70.583,-177.398,8.273,148.857
C05169=1137.785,268.059,-70.613,-177.395,8.276,148.857
C05170=1137.780,268.307,-70.641,-177.392,8.279,148.857
C05171=1137.776,268.556,-70.670,-177.389,8.282,148.857
C05172=1137.772,268.804,-70.699,-177.387,8.285,148.857
C05173=1137.767,269.053,-70.728,-177.384,8.289,148.857
C05174=1137.763,269.300,-70.757,-177.381,8.292,148.857
C05175=1137.759,269.549,-70.785,-177.379,8.295,148.858
C05176=1137.755,269.797,-70.815,-177.376,8.298,148.857
C05177=1137.750,270.045,-70.844,-177.373,8.301,148.857
C05178=1137.745,270.294,-70.873,-177.370,8.305,148.858
C05179=1137.741,270.542,-70.902,-177.367,8.308,148.858
C05180=1137.738,270.790,-70.931,-177.364,8.311,148.857
C05181=1137.733,271.039,-70.960,-177.362,8.314,148.858
C05182=1137.729,271.287,-70.989,-177.359,8.317,148.858
C05183=1137.724,271.534,-71.018,-177.356,8.321,148.858
C05184=1137.720,271.783,-71.048,-177.354,8.324,148.858
C05185=1137.716,272.032,-71.077,-177.351,8.327,148.858
C05186=1137.711,272.280,-71.106,-177.348,8.330,148.858
C05187=1137.707,272.528,-71.135,-177.346,8.333,148.858
C05188=1137.704,272.776,-71.164,-177.342,8.337,148.858
C05189=1137.699,273.024,-71.193,-177.339,8.340,148.858
C05190=1137.695,273.273,-71.222,-177.337,8.343,148.858
C05191=1137.690,273.521,-71.252,-177.334,8.346,148.858
C05192=1137.686,273.769,-71.281,-177.332,8.349,148.858
C05193=1137.682,274.017,-71.310,-177.329,8.353,148.858
C05194=1137.678,274.266,-71.340,-177.326,8.356,148.858
C05195=1137.674,274.514,-71.369,-177.323,8.359,148.858
C05196=1137.669,274.762,-71.399,-177.321,8.362,148.858
C05197=1137.665,275.010,-71.428,-177.317,8.366,148.858
C05198=1137.661,275.258,-71.457,-177.315,8.369,148.858
C05199=1137.656,275.507,-71.486,-177.312,8.372,148.858
C05200=1137.652,275.755,-71.516,-177.309,8.375,148.858
C05201=1137.648,276.003,-71.545,-177.307,8.378,148.858
C05202=1137.644,276.252,-71.574,-177.304,8.382,148.858
C05203=1137.639,276.500,-71.604,-177.301,8.385,148.858
C05204=1137.635,276.748,-71.634,-177.298,8.388,148.858
C05205=1137.631,276.996,-71.664,-177.296,8.391,148.858
C05206=1137.627,277.244,-71.693,-177.293,8.395,148.858
C05207=1137.623,277.492,-71.722,-177.290,8.398,148.858
C05208=1137.618,277.741,-71.752,-177.288,8.401,148.858
C05209=1137.614,277.989,-71.782,-177.285,8.404,148.858
C05210=1137.610,278.238,-71.811,-177.281,8.408,148.858
C05211=1137.605,278.486,-71.841,-177.279,8.411,148.859
C05212=1137.601,278.734,-71.870,-177.276,8.414,148.859
C05213=1137.597,278.982,-71.900,-177.274,8.417,148.859
C05214=1137.593,279.230,-71.930,-177.271,8.421,148.859
C05215=1137.589,279.478,-71.959,-177.268,8.424,148.859
C05216=1137.584,279.727,-71.989,-177.265,8.427,148.859
C05217=1137.580,279.975,-72.019,-177.263,8.430,148.859
C05218=1137.576,280.223,-72.048,-177.260,8.434,148.859
C05219=1137.572,280.471,-72.079,-177.257,8.437,148.859
C05220=1137.568,280.719,-72.108,-177.255,8.441,148.859
C05221=1137.563,280.968,-72.138,-177.252,8.443,148.859
C05222=1137.559,281.216,-72.167,-177.249,8.448,148.859
C05223=1137.555,281.464,-72.198,-177.246,8.450,148.859
C05224=1137.551,281.712,-72.227,-177.244,8.454,148.859
C05225=1137.546,281.961,-72.257,-177.241,8.457,148.859
C05226=1137.542,282.208,-72.287,-177.238,8.461,148.859
C05227=1137.538,282.457,-72.317,-177.235,8.464,148.859
C05228=1137.533,282.705,-72.346,-177.233,8.467,148.860
C05229=1137.529,282.953,-72.377,-177.230,8.471,148.860
C05230=1137.525,283.201,-72.406,-177.227,8.474,148.859
C05231=1137.521,283.449,-72.437,-177.224,8.477,148.860
C05232=1137.516,283.697,-72.467,-177.222,8.480,148.860
C05233=1137.512,283.945,-72.497,-177.219,8.484,148.860
C05234=1137.508,284.193,-72.526,-177.216,8.487,148.860
C05235=1137.503,284.442,-72.557,-177.214,8.490,148.860
C05236=1137.500,284.690,-72.587,-177.211,8.493,148.860
C05237=1137.495,284.938,-72.616,-177.208,8.497,148.860
C05238=1137.491,285.186,-72.647,-177.205,8.500,148.860
C05239=1137.487,285.435,-72.677,-177.203,8.503,148.860
C05240=1137.482,285.683,-72.707,-177.199,8.507,148.860
C05241=1137.478,285.930,-72.737,-177.197,8.510,148.860
C05242=1137.474,286.178,-72.767,-177.195,8.513,148.861
C05243=1137.470,286.427,-72.798,-177.191,8.517,148.861
C05244=1137.466,286.675,-72.827,-177.189,8.520,148.861
C05245=1137.460,286.950,-72.861,-177.186,8.524,148.861
C05246=1137.456,287.226,-72.895,-177.183,8.527,148.861
C05247=1137.451,287.502,-72.929,-177.180,8.531,148.861
C05248=1137.447,287.777,-72.962,-177.177,8.535,148.861
C05249=1137.443,288.026,-72.993,-177.174,8.538,148.861
C05250=1137.438,288.274,-73.023,-177.171,8.542,148.861
C05251=1137.434,288.522,-73.053,-177.168,8.545,148.861
C05252=1137.430,288.770,-73.083,-177.166,8.548,148.861
C05253=1137.425,289.018,-73.114,-177.163,8.552,148.861
C05254=1137.422,289.267,-73.144,-177.160,8.555,148.861
C05255=1137.417,289.515,-73.175,-177.158,8.558,148.861
C05256=1137.413,289.762,-73.205,-177.155,8.562,148.862
C05257=1137.409,290.010,-73.236,-177.152,8.566,148.862
C05258=1137.405,290.259,-73.266,-177.149,8.569,148.862
C05259=1137.400,290.507,-73.296,-177.147,8.573,148.862
C05260=1137.396,290.755,-73.327,-177.144,8.576,148.862
C05261=1137.392,291.003,-73.357,-177.141,8.579,148.862
C05262=1137.388,291.251,-73.388,-177.139,8.582,148.862
C05263=1137.384,291.499,-73.419,-177.136,8.586,148.862
C05264=1137.379,291.747,-73.449,-177.133,8.589,148.862
C05265=1137.375,291.995,-73.479,-177.130,8.593,148.862
C05266=1137.371,292.244,-73.510,-177.128,8.596,148.863
C05267=1137.367,292.492,-73.541,-177.125,8.599,148.863
C05268=1137.363,292.739,-73.571,-177.122,8.603,148.863
C05269=1137.359,292.988,-73.602,-177.120,8.606,148.863
C05270=1137.354,293.236,-73.633,-177.117,8.609,148.863
C05271=1137.350,293.484,-73.663,-177.114,8.613,148.863
C05272=1137.346,293.732,-73.694,-177.111,8.617,148.863
C05273=1137.342,293.980,-73.725,-177.109,8.619,148.863
C05274=1137.338,294.228,-73.755,-177.106,8.624,148.863
C05275=1137.333,294.476,-73.786,-177.103,8.627,148.864
C05276=1137.329,294.725,-73.817,-177.101,8.630,148.864
C05277=1137.325,294.972,-73.847,-177.098,8.634,148.864
C05278=1137.321,295.220,-73.879,-177.095,8.637,148.864
C05279=1137.317,295.468,-73.910,-177.093,8.640,148.864
C05280=1137.312,295.716,-73.940,-177.090,8.644,148.864
C05281=1137.309,295.965,-73.971,-177.087,8.647,148.864
C05282=1137.304,296.213,-74.002,-177.084,8.651,148.864
C05283=1137.300,296.461,-74.032,-177.082,8.654,148.864
C05284=1137.296,296.709,-74.064,-177.079,8.657,148.864
C05285=1137.291,296.957,-74.095,-177.076,8.661,148.865
C05286=1137.288,297.205,-74.126,-177.074,8.665,148.865
C05287=1137.284,297.453,-74.156,-177.071,8.668,148.865
C05288=1137.279,297.701,-74.187,-177.068,8.672,148.865
C05289=1137.275,297.949,-74.219,-177.065,8.675,148.865
C05290=1137.271,298.197,-74.250,-177.063,8.679,148.865
C05291=1137.267,298.445,-74.281,-177.060,8.682,148.865
C05292=1137.263,298.693,-74.311,-177.057,8.685,148.865
C05293=1137.258,298.940,-74.343,-177.054,8.689,148.866
C05294=1137.254,299.189,-74.374,-177.052,8.692,148.866
C05295=1137.250,299.437,-74.404,-177.049,8.695,148.866
C05296=1137.246,299.685,-74.436,-177.046,8.699,148.866
C05297=1137.241,299.933,-74.467,-177.044,8.703,148.866
C05298=1137.238,300.181,-74.499,-177.041,8.706,148.866
C05299=1137.233,300.429,-74.530,-177.038,8.710,148.866
C05300=1137.229,300.678,-74.561,-177.036,8.713,148.867
C05301=1137.225,300.925,-74.592,-177.033,8.717,148.867
C05302=1137.221,301.174,-74.623,-177.030,8.720,148.867
C05303=1137.217,301.421,-74.655,-177.027,8.724,148.867
C05304=1137.212,301.669,-74.686,-177.025,8.727,148.867
C05305=1137.208,301.917,-74.717,-177.023,8.730,148.867
C05306=1137.204,302.165,-74.748,-177.019,8.734,148.867
C05307=1137.200,302.413,-74.780,-177.017,8.737,148.867
C05308=1137.195,302.661,-74.811,-177.014,8.741,148.868
C05309=1137.192,302.909,-74.843,-177.012,8.745,148.868
C05310=1137.187,303.157,-74.873,-177.008,8.748,148.868
C05311=1137.183,303.405,-74.905,-177.006,8.752,148.868
C05312=1137.179,303.654,-74.936,-177.004,8.755,148.868
C05313=1137.175,303.901,-74.968,-177.001,8.759,148.868
C05314=1137.171,304.149,-75.000,-176.998,8.762,148.868
C05315=1137.167,304.397,-75.031,-176.995,8.766,148.869
C05316=1137.163,304.645,-75.062,-176.993,8.769,148.869
C05317=1137.159,304.892,-75.094,-176.990,8.773,148.869
C05318=1137.155,305.141,-75.125,-176.987,8.777,148.869
C05319=1137.150,305.389,-75.157,-176.985,8.780,148.869
C05320=1137.146,305.637,-75.189,-176.982,8.784,148.869
C05321=1137.142,305.885,-75.220,-176.979,8.787,148.869
C05322=1137.138,306.133,-75.252,-176.976,8.791,148.870
C05323=1137.134,306.381,-75.283,-176.974,8.794,148.870
C05324=1137.129,306.628,-75.315,-176.971,8.798,148.870
C05325=1137.125,306.877,-75.347,-176.968,8.801,148.870
C05326=1137.121,307.125,-75.378,-176.966,8.804,148.870
C05327=1137.117,307.372,-75.410,-176.963,8.809,148.870
C05328=1137.113,307.620,-75.442,-176.961,8.812,148.871
C05329=1137.109,307.868,-75.473,-176.958,8.816,148.871
C05330=1137.104,308.117,-75.505,-176.955,8.819,148.871
C05331=1137.100,308.365,-75.537,-176.952,8.823,148.871
C05332=1137.096,308.612,-75.568,-176.950,8.826,148.871
C05333=1137.092,308.860,-75.600,-176.947,8.830,148.871
C05334=1137.088,309.109,-75.633,-176.944,8.833,148.872
C05335=1137.083,309.356,-75.664,-176.941,8.837,148.872
C05336=1137.080,309.604,-75.696,-176.939,8.841,148.872
C05337=1137.076,309.852,-75.728,-176.937,8.844,148.872
C05338=1137.071,310.100,-75.760,-176.934,8.848,148.872
C05339=1137.067,310.348,-75.792,-176.931,8.851,148.873
C05340=1137.064,310.596,-75.823,-176.928,8.855,148.873
C05341=1137.059,310.843,-75.856,-176.926,8.858,148.873
C05342=1137.055,311.091,-75.887,-176.923,8.862,148.873
C05343=1137.051,311.339,-75.919,-176.920,8.866,148.873
C05344=1137.047,311.588,-75.952,-176.918,8.870,148.873
C05345=1137.042,311.835,-75.983,-176.915,8.873,148.874
C05346=1137.039,312.083,-76.015,-176.912,8.877,148.874
C05347=1137.034,312.331,-76.047,-176.910,8.880,148.874
C05348=1137.030,312.579,-76.079,-176.907,8.884,148.874
C05349=1137.026,312.857,-76.115,-176.904,8.888,148.874
C05350=1137.021,313.135,-76.151,-176.901,8.892,148.875
C05351=1137.016,313.413,-76.187,-176.898,8.897,148.875
C05352=1137.012,313.691,-76.224,-176.895,8.901,148.875
C05353=1137.008,313.939,-76.256,-176.892,8.904,148.875
C05354=1137.004,314.187,-76.287,-176.890,8.908,148.875
C05355=1136.999,314.435,-76.320,-176.887,8.911,148.875
C05356=1136.996,314.682,-76.352,-176.884,8.915,148.876
C05357=1136.991,314.931,-76.385,-176.882,8.918,148.876
C05358=1136.988,315.179,-76.416,-176.879,8.922,148.876
C05359=1136.983,315.426,-76.449,-176.877,8.926,148.876
C05360=1136.979,315.674,-76.481,-176.874,8.930,148.876
C05361=1136.975,315.922,-76.514,-176.871,8.933,148.877
C05362=1136.971,316.170,-76.546,-176.868,8.937,148.877
C05363=1136.967,316.418,-76.579,-176.866,8.940,148.877
C05364=1136.963,316.665,-76.610,-176.863,8.944,148.877
C05365=1136.958,316.913,-76.643,-176.861,8.947,148.877
C05366=1136.955,317.161,-76.675,-176.858,8.952,148.878
C05367=1136.950,317.409,-76.707,-176.855,8.955,148.878
C05368=1136.947,317.657,-76.740,-176.853,8.959,148.878
C05369=1136.942,317.905,-76.772,-176.850,8.962,148.878
C05370=1136.938,318.153,-76.806,-176.847,8.966,148.879
C05371=1136.934,318.400,-76.837,-176.844,8.970,148.879
C05372=1136.930,318.648,-76.870,-176.842,8.974,148.879
C05373=1136.926,318.896,-76.902,-176.839,8.978,148.879
C05374=1136.922,319.144,-76.935,-176.837,8.981,148.879
C05375=1136.918,319.392,-76.968,-176.834,8.985,148.880
C05376=1136.914,319.640,-77.000,-176.832,8.988,148.880
C05377=1136.910,319.888,-77.033,-176.829,8.993,148.880
C05378=1136.906,320.136,-77.066,-176.827,8.996,148.880
C05379=1136.902,320.384,-77.098,-176.824,9.000,148.881
C05380=1136.898,320.631,-77.131,-176.821,9.003,148.881
C05381=1136.894,320.879,-77.164,-176.818,9.007,148.881
C05382=1136.890,321.127,-77.196,-176.816,9.010,148.881
C05383=1136.885,321.374,-77.229,-176.813,9.015,148.881
C05384=1136.881,321.622,-77.262,-176.810,9.019,148.882
C05385=1136.877,321.870,-77.294,-176.808,9.022,148.882
C05386=1136.873,322.118,-77.327,-176.805,9.026,148.882
C05387=1136.869,322.365,-77.360,-176.803,9.029,148.882
C05388=1136.865,322.614,-77.392,-176.800,9.034,148.883
C05389=1136.861,322.861,-77.425,-176.798,9.037,148.883
C05390=1136.857,323.109,-77.458,-176.795,9.041,148.883
C05391=1136.853,323.357,-77.491,-176.792,9.044,148.883
C05392=1136.849,323.605,-77.524,-176.789,9.048,148.884
C05393=1136.845,323.852,-77.556,-176.787,9.052,148.884
C05394=1136.841,324.100,-77.589,-176.784,9.056,148.884
C05395=1136.837,324.348,-77.623,-176.781,9.060,148.884
C05396=1136.833,324.596,-77.656,-176.779,9.063,148.885
C05397=1136.828,324.844,-77.688,-176.776,9.067,148.885
C05398=1136.824,325.092,-77.721,-176.774,9.070,148.885
C05399=1136.821,325.339,-77.754,-176.771,9.075,148.885
C05400=1136.817,325.587,-77.787,-176.768,9.079,148.885
C05401=1136.813,325.835,-77.821,-176.766,9.082,148.886
C05402=1136.809,326.083,-77.854,-176.763,9.086,148.886
C05403=1136.805,326.331,-77.887,-176.761,9.090,148.886
C05404=1136.801,326.578,-77.920,-176.758,9.094,148.886
C05405=1136.797,326.788,-77.947,-176.756,9.097,148.887
C05406=1136.793,326.998,-77.976,-176.753,9.100,148.887
C05407=1136.791,327.208,-78.004,-176.751,9.103,148.887
C05408=1136.774,328.262,-78.148,-177.582,10.718,149.518
C05409=1136.770,328.510,-78.181,-177.579,10.720,149.518
C05410=1136.765,328.758,-78.215,-177.576,10.723,149.518
C05411=1136.761,329.005,-78.249,-177.573,10.726,149.518
C05412=1136.757,329.253,-78.282,-177.569,10.728,149.518
C05413=1136.753,329.501,-78.315,-177.567,10.731,149.518
C05414=1136.749,329.749,-78.349,-177.563,10.733,149.517
C05415=1136.745,329.996,-78.382,-177.560,10.736,149.517
C05416=1136.741,330.244,-78.417,-177.557,10.738,149.517
C05417=1136.737,330.492,-78.450,-177.554,10.740,149.517
C05418=1136.733,330.740,-78.483,-177.551,10.743,149.517
C05419=1136.729,330.987,-78.517,-177.548,10.745,149.516
C05420=1136.725,331.235,-78.550,-177.544,10.747,149.516
C05421=1136.721,331.483,-78.585,-177.541,10.750,149.516
C05422=1136.717,331.731,-78.618,-177.538,10.753,149.516
C05423=1136.713,331.978,-78.652,-177.535,10.755,149.516
C05424=1136.709,332.225,-78.685,-177.531,10.758,149.515
C05425=1136.705,332.474,-78.720,-177.528,10.760,149.515
C05426=1136.701,332.721,-78.754,-177.525,10.763,149.515
C05427=1136.697,332.968,-78.787,-177.522,10.765,149.515
C05428=1136.693,333.217,-78.822,-177.519,10.768,149.514
C05429=1136.689,333.464,-78.855,-177.516,10.771,149.514
C05430=1136.685,333.711,-78.889,-177.512,10.773,149.514
C05431=1136.682,333.959,-78.923,-177.509,10.775,149.514
C05432=1136.677,334.207,-78.957,-177.506,10.778,149.514
C05433=1136.670,334.625,-79.015,-177.500,10.782,149.513
C05434=1136.664,335.042,-79.071,-177.494,10.787,149.513
C05435=1136.657,335.459,-79.129,-177.489,10.790,149.513
C05436=1136.650,335.877,-79.186,-177.484,10.795,149.512
C05437=1136.646,336.125,-79.221,-177.480,10.797,149.512
C05438=1136.642,336.372,-79.255,-177.478,10.800,149.512
C05439=1136.639,336.619,-79.289,-177.474,10.803,149.512
C05440=1136.634,336.868,-79.323,-177.471,10.805,149.512
C05441=1136.631,337.115,-79.357,-177.468,10.807,149.511
C05442=1136.627,337.363,-79.391,-177.465,10.810,149.511
C05443=1136.623,337.610,-79.425,-177.461,10.813,149.511
C05444=1136.618,337.857,-79.460,-177.458,10.815,149.511
C05445=1136.615,338.105,-79.494,-177.455,10.818,149.511
C05446=1136.611,338.352,-79.528,-177.451,10.820,149.510
C05447=1136.607,338.600,-79.563,-177.449,10.823,149.510
C05448=1136.603,338.848,-79.596,-177.445,10.825,149.510
C05449=1136.598,339.096,-79.630,-177.442,10.828,149.510
C05450=1136.594,339.344,-79.665,-177.439,10.830,149.510
C05451=1136.591,339.591,-79.699,-177.435,10.833,149.509
C05452=1136.587,339.839,-79.734,-177.432,10.835,149.509
C05453=1136.583,340.086,-79.768,-177.429,10.838,149.509
C05454=1136.579,340.334,-79.803,-177.426,10.840,149.509
C05455=1136.575,340.581,-79.836,-177.422,10.843,149.509
C05456=1136.571,340.829,-79.871,-177.419,10.845,149.508
C05457=1136.567,341.076,-79.905,-177.416,10.848,149.508
C05458=1136.563,341.325,-79.940,-177.412,10.850,149.508
C05459=1136.559,341.571,-79.975,-177.410,10.853,149.508
C05460=1136.555,341.818,-80.009,-177.406,10.855,149.508
C05461=1136.551,342.067,-80.044,-177.403,10.858,149.507
C05462=1136.547,342.314,-80.078,-177.400,10.860,149.507
C05463=1136.543,342.562,-80.113,-177.396,10.863,149.507
C05464=1136.539,342.809,-80.147,-177.393,10.865,149.507
C05465=1136.535,343.057,-80.182,-177.390,10.868,149.507
C05466=1136.531,343.304,-80.216,-177.387,10.870,149.506
C05467=1136.527,343.552,-80.251,-177.383,10.873,149.506
C05468=1136.523,343.800,-80.286,-177.380,10.875,149.506
C05469=1136.520,344.047,-80.320,-177.377,10.878,149.506
C05470=1136.516,344.295,-80.355,-177.373,10.880,149.505
C05471=1136.511,344.542,-80.390,-177.371,10.882,149.505
